# B&R Automation Studio project AutoCon2021 (part 2)

### GlobalTypes.typ
```iecst
(*Main System Interface Types*)

TYPE
	MainIfTyp : 	STRUCT
		Cmd : MainIfCmdTyp;
		Par : MainIfParTyp;
		Cfg : MainIfCfgTyp;
		Status : MainIfStatusTyp;
	END_STRUCT;
	MainIfCmdTyp : 	STRUCT
		Power : BOOL;
		Start : BOOL;
		Stop : BOOL;
		Reset : BOOL;
	END_STRUCT;
	MainIfParTyp : 	STRUCT
		Tmp : USINT;
	END_STRUCT;
	MainIfCfgTyp : 	STRUCT
		ShuttleCount : USINT;
	END_STRUCT;
	MainIfStatusTyp : 	STRUCT
		PowerOn : BOOL;
		Running : BOOL;
		Error : BOOL;
	END_STRUCT;
END_TYPE

(*Process Info Interface*)

TYPE
	ProcessInfoIfTyp : 	STRUCT
		Cmd : ProcessInfoIfCmdTyp;
		Par : ProcessInfoIfParTyp;
		Sts : ProcessInfoIfStsTyp;
	END_STRUCT;
	ProcessInfoIfCmdTyp : 	STRUCT
		Enable : BOOL;
		ResetData : BOOL;
	END_STRUCT;
	ProcessInfoIfParTyp : 	STRUCT
		CurrentProductCount : UDINT;
		CurrentPowderCount : UDINT;
	END_STRUCT;
	ProcessInfoIfStsTyp : 	STRUCT
		Enabled : BOOL;
		CurrentPPM : REAL;
		CurrentPPH : REAL;
		CurrentBlistersPerMinute : REAL;
		CurrentLayersPerMinute : REAL;
	END_STRUCT;
END_TYPE

(*Shuttle Interface Types*)

TYPE
	gShuttleIfTyp : 	STRUCT  (*Interface for controlling a shuttle*)
		Cmd : gShuttleIfCmdTyp; (*Commands to issue to a shuttle*)
		Par : gShuttleIfParTyp; (*Parameters for the process for this shuttle*)
		Cfg : gShuttleIfConfigTyp; (*Configuration values for this shuttle*)
		Flags : USINT;
		Status : gShuttleIfStatusTyp; (*Status information related to this shuttle*)
	END_STRUCT;
	gShuttleIfCmdTyp : 	STRUCT  (*Commands for controlling a shuttle*)
		Enable : BOOL; (*Command for enabling the control of a shuttle in the process*)
		Recover : BOOL; (*Command for a shuttle to start recovery*)
		NextStep : BOOL; (*Command for a shuttle to start the next step in the process*)
		ResetProductInfo : BOOL; (*Command to reset all the product info on a shuttle*)
		Stop : BOOL; (*Command to stop the process for a shuttle*)
	END_STRUCT;
	gShuttleIfParTyp : 	STRUCT  (*Parameters for the shuttle's operation*)
		NumLayers : USINT; (*Number of layers for this defined recipe*)
		MacroIDs : gShuttleIfCfgMacrosTyp; (*Macro's used for routing shuttles*)
	END_STRUCT;
	gShuttleIfCfgMacrosTyp : 	STRUCT  (*Structure of the macro IDs used for operation*)
		LoadToPrintMacroID : gShuttleIfMacroEnum; (*Macro ID used for sending a shuttle from the load station to the print station*)
		PrintToDoseMacroID : gShuttleIfMacroEnum; (*Macro ID used for sending a shuttle from the print station to the Dose station*)
		DoseToPrintMacroID : gShuttleIfMacroEnum; (*Macro ID used for sending a shuttle from the dosing station to the printing station*)
		PrintToTampMacroID : gShuttleIfMacroEnum; (*Macro ID used for sending a shuttle from the printing station to the tamping station*)
		TampToUnloadMacroID : gShuttleIfMacroEnum; (*Macro ID used for sending a shuttle from the tamping station to the unload station*)
		UnloadToLoadMacroID : gShuttleIfMacroEnum; (*Macro ID used for sending a shuttle from the unloading station to the loading station*)
	END_STRUCT;
	gShuttleIfConfigTyp : 	STRUCT  (*Configuration values for a shuttle*)
		ShuttleId : USINT; (*ShuttleID of this shuttle*)
	END_STRUCT;
	gShuttleIfStatusTyp : 	STRUCT  (*Status information for the shuttle*)
		CurrentDestination : gShuttleIfDestEnum; (*Destination the shuttle is currently moving towards*)
		BlisterPresent : BOOL; (*Status flag to denote that a blister pack has been loaded on the shuttle*)
		ProductTamped : BOOL; (*Status flag to denote that the product has  been tamped*)
		CurrentLayer : USINT; (*Current Layer being built on the shuttle*)
		ShuttleInfo : Acp6DShuttleInfoType; (*CurrentStatus Information about the shuttle*)
		Error : BOOL; (*Shuttle is currently in an error state*)
		ErrorState : ShStateEnum; (*State the shuttle errored at*)
		Recovered : BOOL; (*Shuttle has been recovered*)
	END_STRUCT;
	gShuttleIfMacroEnum :
		( (*Macro IDs that are used to denote which macro means what*)
		MACRO_LOAD_TO_PRINT := 128, (*Macro ID used for sending a shuttle from the load station to the print station*)
		MACRO_PRINT_TO_DOSE1, (*Macro ID for moving from the print station to the dose 1 station*)
		MACRO_PRINT_TO_DOSE2, (*Macro ID for moving from the print station to the dose 2 station*)
		MACRO_DOSE_TO_PRINT, (*Macro ID used for sending a shuttle from the dosing station to the printing station*)
		MACRO_PRINT_TO_TAMP, (*Macro ID used for sending a shuttle from the printing station to the tamping station*)
		MACRO_TAMP_TO_UNLOAD, (*Macro ID used for sending a shuttle from the tamping station to the unload station*)
		MACRO_UNLOAD_TO_LOAD, (*Macro ID used for sending a shuttle from the unloading station to the loading station*)
		MACRO_RECOVERY_GROUP0, (*Macro ID used for recovering the group 0 shuttles*)
		MACRO_RECOVERY_GROUP1, (*Macro ID used for recovering the group 1 shuttles*)
		MACRO_RECOVERY_GROUP2 (*Macro ID used for recovering the group 2 shuttles*)
		);
	gShuttleIfDestEnum :
		( (*Destinations for a shuttle to move to*)
		DEST_LOAD, (*Destination Load station*)
		DEST_PRINT, (*Destination Printing station*)
		DEST_DOSE1, (*Destination Dose 1 station*)
		DEST_DOSE2, (*Destination Dose 2 station*)
		DEST_TAMP, (*Destination Tamping station*)
		DEST_UNLOAD (*Destination unload*)
		);
	ShStateEnum :
		(
		SH_OFF, (*Shuttle is in the off/idle state*)
		SH_INIT, (*Shuttle is in the initilization state*)
		SH_STARTUP, (*Shuttle is in the startup state*)
		SH_IDLE, (*Shuttle is in the idle state after having been recovered*)
		SH_MOVE_TO_LOAD, (*Shuttle is moving to the load position*)
		SH_LOAD, (*Shuttle is currently being loaded*)
		SH_MOVE_TO_PRINT, (*Shuttle is moving to the print position*)
		SH_PRINT, (*Shuttle is currently being printed*)
		SH_DECIDE_DOSE, (*Shuttle is deciding which dose station to send the shuttle to*)
		SH_MOVE_TO_DOSE, (*Shuttle is moving towards the defined dosing station*)
		SH_DOSE, (*Shuttle is currently going through the dosing procedure*)
		SH_MOVE_TO_TAMP, (*Shuttle is moving to the tamping location*)
		SH_TAMP, (*Shuttle is currently being tamped*)
		SH_MOVE_TO_OFFLOAD, (*Shuttle is moving to the offload position*)
		SH_OFFLOAD, (*Shuttle is currently being offloaded*)
		SH_ERROR := 65535 (*Shuttle is in the error state*)
		);
END_TYPE

(*6D Controller Interface Types*)

TYPE
	Acp6DCmdType : 	STRUCT
		Power : BOOL;
		ErrorReset : BOOL;
		GetErrorInfo : BOOL;
	END_STRUCT;
	Acp6DCtrlType : 	STRUCT
		Cmd : Acp6DCmdType;
		Status : Acp6DStatusType;
		Par : Acp6DParType;
	END_STRUCT;
	Acp6DParType : 	STRUCT
		Mode : McAcp6DMoveModeEnum;
		PathType : McAcp6DInPlaneMovePathEnum;
		Acceleration : REAL;
		EndVelocity : REAL;
		Velocity : REAL;
		ShuttleID : USINT;
		SegmentID : USINT;
		PositionX : REAL;
		PositionY : REAL;
	END_STRUCT;
	Acp6DStatusType : 	STRUCT
		Error : BOOL;
		ErrorID : DINT;
		Ready : BOOL;
		PowerOn : BOOL;
		ReadyToPowerOn : BOOL;
		ErrorCodes : ARRAY[0..8]OF DINT;
	END_STRUCT;
	Acp6DShuttleInfoType : 	STRUCT
		State : Acp6DShuttleStateInfoTyp;
		Force : Acp6DShuttleForceInfoTyp;
		Position : Acp6DShuttlePosInfoTyp;
	END_STRUCT;
	Acp6DShuttleStateInfoTyp : 	STRUCT
		Valid : BOOL;
		Value : McAcp6DShuttleStateEnum;
	END_STRUCT;
	Acp6DShuttlePosInfoTyp : 	STRUCT
		Valid : BOOL;
		Value : McAcp6DShPositionInfoType;
	END_STRUCT;
	Acp6DShuttleForceInfoTyp : 	STRUCT
		Valid : BOOL;
		Value : McAcp6DShForceInfoType;
	END_STRUCT;
END_TYPE

(*Recovery Interface Type*)

TYPE
	Acp6DRecoveryIfTyp : 	STRUCT
		Cmd : Acp6DRecoveryCmdTyp;
		Par : Acp6DRecoveryParTyp;
		Sts : Acp6DRecoveryStsTyp;
	END_STRUCT;
	Acp6DRecoveryCmdTyp : 	STRUCT
		Recover : BOOL;
		Reset : BOOL;
	END_STRUCT;
	Acp6DRecoveryParTyp : 	STRUCT
		AutoDrivePositions : ARRAY[0..MAX_SHUTTLE_COUNT_ARRAY]OF Acp6DAutoDrivePosTyp;
		Vel : REAL;
		Accel : REAL;
	END_STRUCT;
	Acp6DRecoveryStsTyp : 	STRUCT
		Recovering : BOOL;
		ReadyToStartProc : BOOL;
		Done : BOOL;
		ShuttlesRecovered : BOOL;
		Error : BOOL;
	END_STRUCT;
	Acp6DAutoDrivePosTyp : 	STRUCT
		ShIdx : USINT;
		GroupNum : USINT; (*Group ID used for recovery. Lower group, lower priority*)
		X : REAL;
		Y : REAL;
	END_STRUCT;
END_TYPE

(***********************Station Types*)

TYPE
	StationIfTyp : 	STRUCT
		Cmd : StationIfCmdTyp; (*Commands to a station*)
		Par : {REDUND_UNREPLICABLE} UDINT; (*Address of the parameter structure*)
		Cfg : StationIfCfgTyp; (*Configuration values for the station*)
		Sts : StationIfStsTyp; (*Status of the station*)
	END_STRUCT;
	StationIfCmdTyp : 	STRUCT
		Enable : BOOL; (*Enables the process station*)
		Process : BOOL; (*Start a process for the station with the defined shuttle index*)
		Reset : BOOL; (*Resets the process from an any state*)
	END_STRUCT;
	StationIfCfgTyp : 	STRUCT
		StationPos : StationPositionTyp; (*Station's center world position*)
	END_STRUCT;
	StationIfStsTyp : 	STRUCT
		Enabled : BOOL; (*Signal denoting the station is enabled and in an operational state*)
		Processing : BOOL; (*Signal denoting the station is currently operating on a shuttle*)
		Done : BOOL; (*Signal denoting the current operation has completed*)
		ReadyForNewShuttle : BOOL; (*Signal denoting the station is ready for a new shuttle*)
		Error : BOOL; (*Signal denoting the station has an error present*)
	END_STRUCT;
END_TYPE

(*Load Station Types*)

TYPE
	LoadStationIfTyp : 	STRUCT
		Cmd : LoadStationCmdTyp; (*Commands to the station*)
		Par : LoadStationParTyp; (*Paramters for the station's operation*)
		Cfg : LoadStationCfgTyp; (*Configuration values for the station*)
		Status : LoadStationStatusTyp; (*Status of the station*)
	END_STRUCT;
	LoadStationCmdTyp : 	STRUCT
		Enable : BOOL; (*Enables the process station*)
		Process : BOOL; (*Start a process for the station with the defined shuttle index*)
		Reset : BOOL; (*Resets the process from an any state*)
	END_STRUCT;
	LoadStationParTyp : 	STRUCT
		ShuttleIdx : USINT; (*Index in the gShuttle array for the shuttle in question*)
		WaitTime : TIME; (*Amount of time to wait for the load process*)
	END_STRUCT;
	LoadStationCfgTyp : 	STRUCT
		StationPos : StationPositionTyp; (*Station's center world position*)
	END_STRUCT;
	LoadStationStatusTyp : 	STRUCT
		Enabled : BOOL; (*Signal denoting the station is enabled and in an operational state*)
		Processing : BOOL; (*Signal denoting the station is currently operating on a shuttle*)
		Done : BOOL; (*Signal denoting the current operation has completed*)
		ReadyForNewShuttle : BOOL; (*Signal denoting the station is ready for a new shuttle*)
		Error : BOOL; (*Signal denoting the station has an error present*)
	END_STRUCT;
	StationPositionTyp : 	STRUCT
		X : REAL; (*Station's Global X position*)
		Y : REAL; (*Station's Global Y position*)
	END_STRUCT;
END_TYPE

(*Unload Station Types*)

TYPE
	UnloadStationIfTyp : 	STRUCT
		Cmd : UnloadStationCmdTyp; (*Commands to the station*)
		Par : UnloadStationParTyp; (*Paramters for the station's operation*)
		Cfg : UnloadStationCfgTyp; (*Configuration values for the station*)
		Status : UnloadStationStatusTyp; (*Status of the station*)
	END_STRUCT;
	UnloadStationCmdTyp : 	STRUCT
		Enable : BOOL; (*Enables the process station*)
		Process : BOOL; (*Start a process for the station with the defined shuttle index*)
		Reset : BOOL; (*Resets the process from an any state*)
	END_STRUCT;
	UnloadStationParTyp : 	STRUCT
		ShuttleIdx : USINT; (*Index in the gShuttle array for the shuttle in question*)
		WaitTime : TIME; (*Amount of time to wait for the load process*)
	END_STRUCT;
	UnloadStationCfgTyp : 	STRUCT
		StationPos : StationPositionTyp; (*Station's center world position*)
	END_STRUCT;
	UnloadStationStatusTyp : 	STRUCT
		Enabled : BOOL; (*Signal denoting the station is enabled and in an operational state*)
		Processing : BOOL; (*Signal denoting the station is currently operating on a shuttle*)
		Done : BOOL; (*Signal denoting the current operation has completed*)
		ReadyForNewShuttle : BOOL; (*Signal denoting the station is ready for a new shuttle*)
		Error : BOOL; (*Signal denoting the station has an error present*)
	END_STRUCT;
END_TYPE

(*Print Station Types*)

TYPE
	PrintStationIfTyp : 	STRUCT
		Cmd : PrintStationCmdTyp; (*Commands to the station*)
		Par : PrintStationParTyp; (*Paramters for the station's operation*)
		Cfg : PrintStationCfgTyp; (*Configuration values for the station*)
		Status : PrintStationStatusTyp; (*Status of the station*)
	END_STRUCT;
	PrintStationCmdTyp : 	STRUCT
		Enable : BOOL; (*Enables the process station*)
		Process : BOOL; (*Start a process for the station with the defined shuttle index*)
		Reset : BOOL; (*Resets the process from an any state*)
	END_STRUCT;
	PrintStationParTyp : 	STRUCT
		ShuttleIdx : USINT; (*Index in the gShuttle array for the shuttle in question*)
		PrintVel : REAL; (*Speed at which to complete the print process m/s*)
		PrintEndVel : REAL; (*Speed at which the shuttle should end the print process at m/s*)
		PrintDistanceX : REAL; (*Distance for how far the print movement will go in the X direction (m)*)
		PrintDistanceY : REAL; (*Distance for how far the print movement will go in the Y direction(m)*)
		PrintAccel : REAL; (*Acceleration at which to use for the print process m/s2*)
	END_STRUCT;
	PrintStationCfgTyp : 	STRUCT
		StationPos : StationPositionTyp; (*Station's center world position*)
	END_STRUCT;
	PrintStationStatusTyp : 	STRUCT
		Enabled : BOOL; (*Signal denoting the station is enabled and in an operational state*)
		ReadyForNewShuttle : BOOL; (*Signal denoting the station is ready for a new shuttle*)
		Processing : BOOL; (*Signal denoting the station is currently operating on a shuttle*)
		Done : BOOL; (*Signal denoting the current operation has completed*)
		Error : BOOL; (*Signal denoting the station has an error present*)
	END_STRUCT;
END_TYPE

(*Dose Station Types*)

TYPE
	DoseStationIfTyp : 	STRUCT
		Cmd : DoseStationCmdTyp; (*Commands to the station*)
		Par : DoseStationParTyp; (*Paramters for the station's operation*)
		Cfg : DoseStationCfgTyp; (*Configuration values for the station*)
		Status : DoseStationStatusTyp; (*Status of the station*)
	END_STRUCT;
	DoseStationCmdTyp : 	STRUCT
		Enable : BOOL; (*Enables the process station*)
		Process : BOOL; (*Start a process for the station with the defined shuttle index*)
		Reset : BOOL; (*Resets the process from an any state*)
	END_STRUCT;
	DoseStationParTyp : 	STRUCT
		ShuttleIdx : USINT; (*Index in the gShuttle array for the shuttle in question*)
		Vel : REAL; (*Velocity to move for the defined index movement*)
		EndVel : REAL; (*Velocity to end the movement at for the defined index movement*)
		Accel : REAL; (*Acceleration to use for the defined index movement*)
		WaitTime : TIME; (*Time needed to preform each dose process*)
		NumRowsOfCavities : USINT; (*Number of rows of the cavities in the blister pack. Will be indexing this many times in the dosing process*)
		SpaceBetweenCavities : DoseIndexMovParsTyp; (*Space between cavities to index through*)
		FirstCavityPosition : DoseIndexMovParsTyp; (*Offset in m for the first cavity*)
	END_STRUCT;
	DoseStationCfgTyp : 	STRUCT
		StationPos : StationPositionTyp; (*Station's center world position*)
	END_STRUCT;
	DoseStationStatusTyp : 	STRUCT
		Enabled : BOOL; (*Signal denoting the station is enabled and in an operational state*)
		ReadyForNewShuttle : BOOL; (*Signal denoting the station is ready for a new shuttle*)
		Processing : BOOL; (*Signal denoting the station is currently operating on a shuttle*)
		Done : BOOL; (*Signal denoting the current operation has completed*)
		Error : BOOL; (*Signal denoting the station has an error present*)
	END_STRUCT;
	DoseIndexMovParsTyp : 	STRUCT
		DistX : REAL; (*Relative distance in X to move for a defined index (m)*)
		DistY : REAL; (*Relative distance in Y to move for a defined index (m)*)
	END_STRUCT;
END_TYPE

(*Tamp Station Types*)

TYPE
	TampStationIfTyp : 	STRUCT
		Cmd : TampStationCmdTyp; (*Commands to the station*)
		Par : TampStationParTyp; (*Paramters for the station's operation*)
		Cfg : TampStationCfgTyp; (*Configuration values for the station*)
		Status : TampStationStatusTyp; (*Status of the station*)
	END_STRUCT;
	TampStationCmdTyp : 	STRUCT
		Enable : BOOL; (*Enables the process station*)
		Process : BOOL; (*Start a process for the station with the defined shuttle index*)
		Reset : BOOL; (*Resets the process from an any state*)
	END_STRUCT;
	TampStationParTyp : 	STRUCT
		ShuttleIdx : USINT; (*Index in the gShuttle array for the shuttle in question*)
		EntranceMovement : TampMovementParTyp; (*Relative position to enter the tamp position*)
		ExitMovement : TampMovementParTyp; (*Relative positions to exit the tamp position*)
		TampHeight : REAL; (*Height in which to preform the z movement for the tamp process (m)*)
		Vel : REAL; (*Velocity to move for the defined index movement*)
		EndVel : REAL; (*Velocity to end the movement at for the defined index movement*)
		Accel : REAL; (*Acceleration to use for the defined index movement*)
		WaitTime : TIME; (*Time needed to preform each dose process*)
	END_STRUCT;
	TampStationCfgTyp : 	STRUCT
		StationPos : StationPositionTyp; (*Station's center world position*)
	END_STRUCT;
	TampStationStatusTyp : 	STRUCT
		Enabled : BOOL; (*Signal denoting the station is enabled and in an operational state*)
		ReadyForNewShuttle : BOOL; (*Signal denoting the station is ready for a new shuttle*)
		Processing : BOOL; (*Signal denoting the station is currently operating on a shuttle*)
		Done : BOOL; (*Signal denoting the current operation has completed*)
		Error : BOOL; (*Signal denoting the station has an error present*)
	END_STRUCT;
	TampMovementParTyp : 	STRUCT
		DistX : REAL; (*Relative distance in X to move for a defined movement(m)*)
		DistY : REAL; (*Relative distance in Y to move for a defined movement(m)*)
	END_STRUCT;
END_TYPE
```

### Package Logical/Source/ShuttleCtrl - Package that contains code for controlling individual shuttles

### Program Logical/Source/ShuttleCtrl/ShCtrl (IEC)

#### Cyclic.st - Cyclic code
```iecst
PROGRAM _CYCLIC
	FOR i:= 0 TO gMainIf.Cfg.ShuttleCount - 1 DO

		IF gShuttleIf[i].Status.CurrentDestination = DEST_DOSE1 THEN
			pDoseStationIf ACCESS ADR(gDoseStationsIf[0]);
		ELSIF gShuttleIf[i].Status.CurrentDestination = DEST_DOSE2 THEN
			pDoseStationIf ACCESS ADR(gDoseStationsIf[1]);
		END_IF

		CASE shState[i] OF
			SH_OFF:  //******************************************************************************** Shuttle is in the off/idle state
				IF gShuttleIf[i].Cmd.Enable THEN
					shState[i] := SH_INIT;
				ELSE

				END_IF
			SH_INIT:  //******************************************************************************** Shuttle is in the initilization state
				//In this state we could make any checks on the current shuttle process perhaps in order to aide in recovery?

				shState[i] := SH_STARTUP;
			SH_STARTUP:  //******************************************************************************** Shuttle is in the startup state
				//In this state maybe we have triggered recovery and we're waiting for the autodrive to complete
				shState[i] := SH_IDLE;
			SH_IDLE:  //******************************************************************************** Shuttle is in the idle state
				IF gShuttleIf[i].Cmd.NextStep THEN
					gShuttleIf[i].Cmd.NextStep := FALSE;
					//Evaluate the current step to determine what the next step should be
					shFbs[i].ShRunMacroFb.Controller := ADR(gMcAcp6DController);
					shFbs[i].ShRunMacroFb.ShuttleID := gShuttleIf[i].Cfg.ShuttleId;
					shFbs[i].ShRunMacroFb.MacroID := UDINT_TO_USINT(gShuttleIf[i].Par.MacroIDs.UnloadToLoadMacroID);
					shFbs[i].ShRunMacroFb.Execute := TRUE;
					gShuttleIf[i].Status.CurrentDestination := DEST_LOAD;
					LogDebug(gAuditTrail,i,"Sent to Load");
					//MpAuditCustomEvent(gAuditTrail,"INFO","Sh","Powered On");

					shState[i] := SH_MOVE_TO_LOAD;
				END_IF
			SH_MOVE_TO_LOAD:  //******************************************************************************** Shuttle is moving to the load position
				IF shFbs[i].ShRunMacroFb.Error THEN
					gShuttleIf[i].Status.Error := TRUE;
					gShuttleIf[i].Status.ErrorState := shState[i];
					shState[i] := SH_ERROR;
				ELSIF shFbs[i].ShRunMacroFb.Done AND (gLoadStationIf.Par.ShuttleIdx = STATION_IS_EMPTY AND gLoadStationIf.Status.ReadyForNewShuttle)
					AND PositionValidation(ADR(gLoadStationIf.Cfg.StationPos),ADR(gShuttleIf[i].Status.ShuttleInfo.Position)) THEN
					gLoadStationIf.Par.ShuttleIdx := i;
					gLoadStationIf.Cmd.Process := TRUE;

					LogDebug(gAuditTrail,i,"Arrived at Load");

					shFbs[i].ShRunMacroFb.Execute := FALSE;
					shState[i] := SH_LOAD;
				END_IF
			SH_LOAD:  //******************************************************************************** Shuttle is currently being loaded
				//Station has control on the shuttle during this section
				IF gShuttleIf[i].Cmd.NextStep THEN
					gLoadStationIf.Cmd.Process := FALSE; //Respond to the Load station we're done

					gShuttleIf[i].Status.BlisterPresent := TRUE;
					gShuttleIf[i].Cmd.NextStep := FALSE;
					gShuttleIf[i].Status.CurrentDestination := DEST_PRINT;

					shFbs[i].ShRunMacroFb.Controller := ADR(gMcAcp6DController);
					shFbs[i].ShRunMacroFb.ShuttleID := gShuttleIf[i].Cfg.ShuttleId;
					shFbs[i].ShRunMacroFb.MacroID := UDINT_TO_USINT(gShuttleIf[i].Par.MacroIDs.LoadToPrintMacroID);
					shFbs[i].ShRunMacroFb.Execute := TRUE;

					LogDebug(gAuditTrail,i,"Sent To Print");

					shState[i] := SH_MOVE_TO_PRINT;
				END_IF
			SH_MOVE_TO_PRINT:  //******************************************************************************** Shuttle is moving to the print position
				IF shFbs[i].ShRunMacroFb.Error THEN
					gShuttleIf[i].Status.Error := TRUE;
					gShuttleIf[i].Status.ErrorState := shState[i];
					shState[i] := SH_ERROR;
				ELSIF shFbs[i].ShRunMacroFb.Done AND (gPrintStationIf.Par.ShuttleIdx = STATION_IS_EMPTY AND gPrintStationIf.Status.ReadyForNewShuttle)
					AND PositionValidation(ADR(gPrintStationIf.Cfg.StationPos),ADR(gShuttleIf[i].Status.ShuttleInfo.Position)) THEN
					gPrintStationIf.Par.ShuttleIdx := i; //Replace with idx when adding the loop
					gPrintStationIf.Cmd.Process := TRUE;

					LogDebug(gAuditTrail,i,"Arrived at Print");

					shFbs[i].ShRunMacroFb.Execute := FALSE;
					shState[i] := SH_PRINT;
				END_IF
			SH_PRINT:  //******************************************************************************** Shuttle is currently being printed
				//Station has control on the shuttle during this section
				IF gShuttleIf[i].Cmd.NextStep THEN
					gPrintStationIf.Cmd.Process := FALSE; //Respond to the print station we're done

					gShuttleIf[i].Status.CurrentLayer :=  gShuttleIf[i].Status.CurrentLayer + 1;
					LogDebug(gAuditTrail,i,"Print complete");
					gShuttleIf[i].Cmd.NextStep := FALSE;

					shState[i] := SH_DECIDE_DOSE;
				END_IF
			SH_DECIDE_DOSE:  //******************************************************************************** Shuttle is deciding which dose station to send the shuttle to
				//First check if the layers have finished
				IF gShuttleIf[i].Status.CurrentLayer > gShuttleIf[i].Par.NumLayers THEN
					//We've finished layering move to the tamp state
					shFbs[i].ShRunMacroFb.Controller := ADR(gMcAcp6DController);
					shFbs[i].ShRunMacroFb.ShuttleID := gShuttleIf[i].Cfg.ShuttleId;
					shFbs[i].ShRunMacroFb.MacroID := UDINT_TO_USINT(gShuttleIf[i].Par.MacroIDs.PrintToTampMacroID);
					shFbs[i].ShRunMacroFb.Execute := TRUE;

					gShuttleIf[i].Status.CurrentDestination := DEST_TAMP;
					LogDebug(gAuditTrail,i,"Sent to Tamp");

					shState[i] := SH_MOVE_TO_TAMP;
				ELSE
					//Need to determine which doser is available
					IF NextDoseStation = DEST_DOSE1 THEN
						gShuttleIf[i].Par.MacroIDs.PrintToDoseMacroID := MACRO_PRINT_TO_DOSE1;
						gShuttleIf[i].Status.CurrentDestination := DEST_DOSE1;
						LogDebug(gAuditTrail,i,"Sent To Dose 1");
						NextDoseStation := DEST_DOSE2;
					ELSE
						gShuttleIf[i].Par.MacroIDs.PrintToDoseMacroID := MACRO_PRINT_TO_DOSE2;
						gShuttleIf[i].Status.CurrentDestination := DEST_DOSE2;
						LogDebug(gAuditTrail,i,"Sent To Dose 2");
						NextDoseStation := DEST_DOSE1;
					END_IF

					shFbs[i].ShRunMacroFb.Controller := ADR(gMcAcp6DController);
					shFbs[i].ShRunMacroFb.ShuttleID := gShuttleIf[i].Cfg.ShuttleId;
					shFbs[i].ShRunMacroFb.MacroID := UDINT_TO_USINT(gShuttleIf[i].Par.MacroIDs.PrintToDoseMacroID);
					shFbs[i].ShRunMacroFb.Execute := TRUE;

					shState[i] := SH_MOVE_TO_DOSE;
				END_IF
			SH_MOVE_TO_DOSE:  //******************************************************************************** Shuttle is moving towards the defined dosing station
				IF shFbs[i].ShRunMacroFb.Error THEN
					gShuttleIf[i].Status.Error := TRUE;
					gShuttleIf[i].Status.ErrorState := shState[i];
					shState[i] := SH_ERROR;
				ELSIF shFbs[i].ShRunMacroFb.Done AND (pDoseStationIf.Par.ShuttleIdx = STATION_IS_EMPTY AND pDoseStationIf.Status.ReadyForNewShuttle AND NOT pDoseStationIf.Cmd.Process)
					AND PositionValidation(ADR(pDoseStationIf.Cfg.StationPos),ADR(gShuttleIf[i].Status.ShuttleInfo.Position)) THEN//Wait for the movement to end and the Station to be ready to accept a new shuttle
					pDoseStationIf.Par.ShuttleIdx := i;
					pDoseStationIf.Cmd.Process := TRUE;

					LogDebug(gAuditTrail,i,"Arrived at Dose");

					shFbs[i].ShRunMacroFb.Execute := FALSE;
					shState[i] := SH_DOSE;
				END_IF
			SH_DOSE:  //******************************************************************************** Shuttle is currently going through the dosing procedure
				//Station has control on the shuttle during this section
				IF gShuttleIf[i].Cmd.NextStep THEN
					gShuttleIf[i].Cmd.NextStep := FALSE;
					pDoseStationIf.Cmd.Process := FALSE; //Respond to the dose station we're done

					gShuttleIf[i].Status.CurrentDestination := DEST_PRINT;

					shFbs[i].ShRunMacroFb.Controller := ADR(gMcAcp6DController);
					shFbs[i].ShRunMacroFb.ShuttleID := gShuttleIf[i].Cfg.ShuttleId;
					shFbs[i].ShRunMacroFb.MacroID := UDINT_TO_USINT(gShuttleIf[i].Par.MacroIDs.DoseToPrintMacroID);
					shFbs[i].ShRunMacroFb.Execute := TRUE;

					LogDebug(gAuditTrail,i,"Sent To Print");

					shState[i] := SH_MOVE_TO_PRINT;
				END_IF
			SH_MOVE_TO_TAMP:  //******************************************************************************** Shuttle is moving to the tamping location
				IF shFbs[i].ShRunMacroFb.Error THEN
					gShuttleIf[i].Status.Error := TRUE;
					gShuttleIf[i].Status.ErrorState := shState[i];
					shState[i] := SH_ERROR;
				ELSIF shFbs[i].ShRunMacroFb.Done AND (gTampStationIf.Par.ShuttleIdx = STATION_IS_EMPTY AND gTampStationIf.Status.ReadyForNewShuttle)
					AND PositionValidation(ADR(gTampStationIf.Cfg.StationPos),ADR(gShuttleIf[i].Status.ShuttleInfo.Position)) THEN
					gTampStationIf.Par.ShuttleIdx := i;
					gTampStationIf.Cmd.Process := TRUE;

					LogDebug(gAuditTrail,i,"Arrived at Tamp");

					shFbs[i].ShRunMacroFb.Execute := FALSE;
					shState[i] := SH_TAMP;
				END_IF
			SH_TAMP:  //******************************************************************************** Shuttle is currently being tamped
				//Station has control on the shuttle during this section
				IF gShuttleIf[i].Cmd.NextStep THEN
					gTampStationIf.Cmd.Process := FALSE;//Respond to the unload station we're done

					gShuttleIf[i].Status.ProductTamped := TRUE;
					gShuttleIf[i].Cmd.NextStep := FALSE;

					gShuttleIf[i].Status.CurrentDestination := DEST_UNLOAD;

					shFbs[i].ShRunMacroFb.Controller := ADR(gMcAcp6DController);
					shFbs[i].ShRunMacroFb.ShuttleID := gShuttleIf[i].Cfg.ShuttleId;
					shFbs[i].ShRunMacroFb.MacroID := UDINT_TO_USINT(gShuttleIf[i].Par.MacroIDs.TampToUnloadMacroID);
					shFbs[i].ShRunMacroFb.Execute := TRUE;

					LogDebug(gAuditTrail,i,"Sent To Unload");

					shState[i] := SH_MOVE_TO_OFFLOAD;
				END_IF
			SH_MOVE_TO_OFFLOAD:  //******************************************************************************** Shuttle is moving to the offload position
				IF shFbs[i].ShRunMacroFb.Error THEN
					gShuttleIf[i].Status.Error := TRUE;
					gShuttleIf[i].Status.ErrorState := shState[i];
					shState[i] := SH_ERROR;
				ELSIF shFbs[i].ShRunMacroFb.Done AND (gUnloadStationIf.Par.ShuttleIdx = STATION_IS_EMPTY AND gUnloadStationIf.Status.ReadyForNewShuttle)
					AND PositionValidation(ADR(gUnloadStationIf.Cfg.StationPos),ADR(gShuttleIf[i].Status.ShuttleInfo.Position)) THEN
					gUnloadStationIf.Par.ShuttleIdx := i;
					gUnloadStationIf.Cmd.Process := TRUE;

					LogDebug(gAuditTrail,i,"Arrived at unload");

					shFbs[i].ShRunMacroFb.Execute := FALSE;
					shState[i] := SH_OFFLOAD;
				END_IF
			SH_OFFLOAD:  //******************************************************************************** Shuttle is currently being offloaded
				//Station has control on the shuttle during this section
				IF gShuttleIf[i].Cmd.NextStep THEN
					gUnloadStationIf.Cmd.Process := FALSE; //Respond to the unload station we're done

					gShuttleIf[i].Cmd.NextStep := FALSE;
					gShuttleIf[i].Cmd.ResetProductInfo := TRUE;
					gShuttleIf[i].Status.CurrentDestination := DEST_LOAD;

					//Increment the process counter
					gProcessInfoIf.Par.CurrentProductCount := gProcessInfoIf.Par.CurrentProductCount + 1;

					IF gShuttleIf[i].Cmd.Stop THEN
						gShuttleIf[i].Cmd.Stop := FALSE;
						shState[i] := SH_INIT;
					ELSE
						shFbs[i].ShRunMacroFb.Controller := ADR(gMcAcp6DController);
						shFbs[i].ShRunMacroFb.ShuttleID := gShuttleIf[i].Cfg.ShuttleId;
						shFbs[i].ShRunMacroFb.MacroID := UDINT_TO_USINT(gShuttleIf[i].Par.MacroIDs.UnloadToLoadMacroID);
						shFbs[i].ShRunMacroFb.Execute := TRUE;

						LogDebug(gAuditTrail,i,"Sent To Load");

						shState[i] := SH_MOVE_TO_LOAD;
					END_IF

				END_IF
			SH_ERROR: //******************************************************************************** Shuttle is in the error state

		END_CASE;
		shFbs[i].ShRunMacroFb();

		IF gShuttleIf[i].Cmd.ResetProductInfo THEN
			gShuttleIf[i].Status.CurrentDestination := DEST_LOAD;
			gShuttleIf[i].Status.BlisterPresent := FALSE;
			gShuttleIf[i].Status.CurrentLayer := 0;
			gShuttleIf[i].Status.Error := FALSE;
			gShuttleIf[i].Status.ErrorState := 0;
			gShuttleIf[i].Status.ProductTamped := 0;
			gShuttleIf[i].Cmd.ResetProductInfo := FALSE;
		END_IF
	END_FOR;
	pDebugIf ACCESS ADR(gShuttleIf[debugIdx]);
	pDebugState ACCESS ADR(shState[debugIdx]);
	pDebugFbs ACCESS ADR(shFbs[debugIdx]);

END_PROGRAM
```

#### Init.st - Init code
```iecst
PROGRAM _INIT
	FOR i:=0 TO MAX_SHUTTLE_COUNT-1 DO
		gShuttleIf[i].Par.MacroIDs.LoadToPrintMacroID := MACRO_LOAD_TO_PRINT;
		gShuttleIf[i].Par.MacroIDs.PrintToTampMacroID := MACRO_PRINT_TO_TAMP;
		gShuttleIf[i].Par.MacroIDs.PrintToDoseMacroID := MACRO_PRINT_TO_DOSE2; //Hard coding this for now
		gShuttleIf[i].Par.MacroIDs.DoseToPrintMacroID:= MACRO_DOSE_TO_PRINT;
		gShuttleIf[i].Par.MacroIDs.TampToUnloadMacroID := MACRO_TAMP_TO_UNLOAD;
		gShuttleIf[i].Par.MacroIDs.UnloadToLoadMacroID := MACRO_UNLOAD_TO_LOAD;
		//The print to dose is defined in the shuttle decide dose task

		gShuttleIf[i].Par.NumLayers := 4;
	END_FOR;

	NextDoseStation := DEST_DOSE1;
END_PROGRAM
```

#### Types.typ - Local data types
```iecst
TYPE
	ShFbsTyp : 	STRUCT
		ShRunMacroFb : MC_BR_MacroRun_Acp6D; (*Execute a macro on the current shuttle*)
	END_STRUCT;
	ShCycleIfs : {REDUND_UNREPLICABLE} 	STRUCT
		Dose : REFERENCE TO DoseStationIfTyp;
	END_STRUCT;
END_TYPE
```

#### Variables.var - Local variables
```iecst
VAR
	i : USINT; (*Loop index*)
	shState : ARRAY[0..MAX_SHUTTLE_COUNT_ARRAY] OF ShStateEnum;
	shFbs : ARRAY[0..MAX_SHUTTLE_COUNT_ARRAY] OF ShFbsTyp;
	stationIfs : {REDUND_UNREPLICABLE} ARRAY[0..MAX_SHUTTLE_COUNT_ARRAY] OF ShCycleIfs;
	NextDoseStation : gShuttleIfDestEnum;
	pDoseStationIf : REFERENCE TO DoseStationIfTyp;
	pDebugIf : REFERENCE TO gShuttleIfTyp;
	pDebugFbs : REFERENCE TO ShFbsTyp;
	pDebugState : REFERENCE TO ShStateEnum;
	debugIdx : USINT;
END_VAR
```

#### LocalFunctions.fun
```iecst
FUNCTION LogDebug : USINT
	VAR_INPUT
		MpLink : MpComIdentType;
		Idx : USINT;
		Msg : WSTRING[100];
	END_VAR
	VAR
		msg : WSTRING[100];
		typ : WSTRING[100];
	END_VAR
END_FUNCTION

{REDUND_ERROR} FUNCTION PositionValidation : BOOL (*Validates if a shuttle is in the defined position*) (*$GROUP=User,$CAT=User,$GROUPICON=User.png,$CATICON=User.png*)
	VAR_INPUT
		DestinationPosition : REFERENCE TO StationPositionTyp;
		CurrentInfo : REFERENCE TO Acp6DShuttlePosInfoTyp;
	END_VAR
END_FUNCTION
```

#### PositionValidation.st
```iecst
(* Validates if a shuttle is in the defined position *)
FUNCTION PositionValidation
	IF CurrentInfo.Valid THEN
		IF CurrentInfo.Value.X >= DestinationPosition.X - 0.00001
			AND CurrentInfo.Value.X <= DestinationPosition.X + 0.00001
			AND CurrentInfo.Value.Y >= DestinationPosition.Y - 0.00001
			AND CurrentInfo.Value.Y <= DestinationPosition.Y + 0.00001 THEN
			PositionValidation := TRUE;
		ELSE
			PositionValidation := FALSE;
		END_IF

	ELSE
		PositionValidation := FALSE;
	END_IF
END_FUNCTION

FUNCTION LogDebug
	msg := "";
	typ := "Sh ";
	typ := USINT_TO_WSTRING(Idx);
	MpAuditCustomEvent(MpLink,"DEBUG",typ,Msg);
END_FUNCTION
```

#### LocalFunctions.st - not listed in the package file held
```iecst
(* Validates if a shuttle is in the defined position *)
FUNCTION PositionValidation
	IF CurrentInfo.Valid THEN
		IF CurrentInfo.Value.X >= DestinationPosition.X - 0.00001
			AND CurrentInfo.Value.X <= DestinationPosition.X + 0.00001
			AND CurrentInfo.Value.Y >= DestinationPosition.Y - 0.00001
			AND CurrentInfo.Value.Y <= DestinationPosition.Y + 0.00001 THEN
			PositionValidation := TRUE;
		ELSE
			PositionValidation := FALSE;
		END_IF

	ELSE
		PositionValidation := FALSE;
	END_IF
END_FUNCTION

FUNCTION LogDebug
	msg := "";
	typ := "Sh ";
	typ := USINT_TO_WSTRING(Idx);
	MpAuditCustomEvent(MpLink,"DEBUG",typ,Msg);
END_FUNCTION

FUNCTION BufferCount
	LaneCounts[0] := 0;
	LaneCounts[1] := 0;
	LaneCounts[2] := 0;
	FOR i:=0 TO ShuttleCnt - 1 DO
		IF Shuttles[i].Sts.ProductInfo.Buffer THEN
			LaneCounts[Shuttles[i].Sts.ProductInfo.BufferLane] := LaneCounts[Shuttles[i].Sts.ProductInfo.BufferLane] + 1;
		END_IF
	END_FOR;
END_FUNCTION

FUNCTION GetNextLane
	lowestCount := 255;
	FOR i := 0 TO 2 DO
		IF LaneCounts[i] < lowestCount THEN
			lowestCount := LaneCounts[i];
			curLane := i;
		END_IF
	END_FOR
	GetNextLane := curLane;
END_FUNCTION
```

### Program Logical/Source/ShuttleCtrl/Recovery (IEC)

#### Types.typ
```iecst
TYPE
	RecoveryFbs : 	STRUCT
		AsyncMoveFb : MC_BR_MoveInPlaneAsync_Acp6D;
		MacroRunFb : ARRAY[0..MAX_SHUTTLE_COUNT_ARRAY]OF MC_BR_MacroRun_Acp6D;
	END_STRUCT;
	RecoveryStateEnum :
		(
		RECOVER_IDLE, (*Recovery is in an idle state*)
		RECOVER_INIT, (*Initalize recovery state*)
		RECOVER_AUTODRIVE, (*Preform autodrive movement for recovery*)
		RECOVER_WAIT_ALL_RECOVER, (*Preform the loop through all shuttles to accomplish the reocvery*)
		RECOVER_DONE, (*Recovery has been completed*)
		RECOVER_ERROR (*Recovery had an error*)
		);
END_TYPE
```

#### Variables.var
```iecst
VAR
	CurrentGroup : USINT;
	GroupRecovered : BOOL;
	state : RecoveryStateEnum;
	RecoverFbs : RecoveryFbs;
END_VAR
VAR CONSTANT
	NUM_GROUPS : USINT := 3;
END_VAR
VAR
	i : USINT;
END_VAR
```

#### Cyclic.st
```iecst
PROGRAM _CYCLIC

	(*
	Shuttle reocvery
		Move all shuttles to autodrive positions
		Wait for autodrive to be finished
		loop through each shuttle
			if that shuttle's group is current
				it is not recovered,
					groupRecovered=false
					Evaluate each shuttle's position
					Send it to the unload position and set the "Next step cmd" to be true
				else
					onwards, do nothing

	*)

	CASE state OF
		RECOVER_IDLE:   //******************************************************************************** Recovery is in an idle state*)
			IF g6DRecoveryIf.Cmd.Recover THEN
				g6DRecoveryIf.Sts.Recovering := TRUE;
				state := RECOVER_INIT;
			END_IF
		RECOVER_INIT:   //******************************************************************************** Initalize recovery state*)
			RecoverFbs.AsyncMoveFb.Controller := ADR(gMcAcp6DController);
			RecoverFbs.AsyncMoveFb.NumberOfShuttles := gMainIf.Cfg.ShuttleCount;
			RecoverFbs.AsyncMoveFb.Velocity := g6DRecoveryIf.Par.Vel;
			RecoverFbs.AsyncMoveFb.Acceleration := g6DRecoveryIf.Par.Accel;
			FOR i:=0 TO gMainIf.Cfg.ShuttleCount - 1 DO
				RecoverFbs.AsyncMoveFb.PositionX[i] := g6DRecoveryIf.Par.AutoDrivePositions[i].X;
				RecoverFbs.AsyncMoveFb.PositionY[i] := g6DRecoveryIf.Par.AutoDrivePositions[i].Y;
				RecoverFbs.AsyncMoveFb.ShuttleID[i] := gShuttleIf[g6DRecoveryIf.Par.AutoDrivePositions[i].ShIdx].Cfg.ShuttleId;
				IF RecoverFbs.AsyncMoveFb.ShuttleID[i] = 0 THEN// Invalid shuttle id here
					g6DRecoveryIf.Sts.Error := TRUE;
				END_IF
			END_FOR;
			IF NOT g6DRecoveryIf.Sts.Error THEN
				RecoverFbs.AsyncMoveFb.Execute := TRUE;
				state := RECOVER_AUTODRIVE;
			ELSE
				state := RECOVER_ERROR;
			END_IF

		RECOVER_AUTODRIVE:   //******************************************************************************** Preform autodrive movement for recovery*)
			IF RecoverFbs.AsyncMoveFb.Error THEN
				g6DRecoveryIf.Sts.Error := TRUE;
				state := RECOVER_ERROR;
			ELSIF RecoverFbs.AsyncMoveFb.Done THEN
				g6DRecoveryIf.Sts.ReadyToStartProc := TRUE;
				RecoverFbs.AsyncMoveFb.Execute := FALSE;

				CurrentGroup := 0;
				state := RECOVER_WAIT_ALL_RECOVER;
			END_IF
		RECOVER_WAIT_ALL_RECOVER:   //******************************************************************************** Preform the loop through all shuttles to accomplish the reocvery*)
			//Ideally this should be in a FB
			GroupRecovered := TRUE;
			FOR i:=0 TO gMainIf.Cfg.ShuttleCount -1 DO
				IF g6DRecoveryIf.Par.AutoDrivePositions[i].GroupNum = CurrentGroup THEN
					IF NOT gShuttleIf[g6DRecoveryIf.Par.AutoDrivePositions[i].ShIdx].Status.Recovered THEN
						GroupRecovered := FALSE;
						IF CurrentGroup = 0 THEN
							gShuttleIf[g6DRecoveryIf.Par.AutoDrivePositions[i].ShIdx].Status.Recovered := TRUE;
							gShuttleIf[g6DRecoveryIf.Par.AutoDrivePositions[i].ShIdx].Cmd.NextStep := TRUE;
						ELSE
							RecoverFbs.MacroRunFb[i].Controller := ADR(gMcAcp6DController);
							RecoverFbs.MacroRunFb[i].MacroID := DINT_TO_USINT(MACRO_RECOVERY_GROUP0) + CurrentGroup;
							RecoverFbs.MacroRunFb[i].ShuttleID := gShuttleIf[g6DRecoveryIf.Par.AutoDrivePositions[i].ShIdx].Cfg.ShuttleId;
							RecoverFbs.MacroRunFb[i].Execute := TRUE;

							IF RecoverFbs.MacroRunFb[i].Error THEN
								g6DRecoveryIf.Sts.Error := TRUE;
							ELSIF RecoverFbs.MacroRunFb[i].Acknowledge THEN
								RecoverFbs.MacroRunFb[i].Execute := FALSE;
								gShuttleIf[g6DRecoveryIf.Par.AutoDrivePositions[i].ShIdx].Cmd.NextStep := TRUE;
								gShuttleIf[g6DRecoveryIf.Par.AutoDrivePositions[i].ShIdx].Status.Recovered := TRUE;
							END_IF
						END_IF
					ELSE
						//Already recovered don't have to do anything

					END_IF
				END_IF
			END_FOR;
			IF GroupRecovered THEN
				CurrentGroup := CurrentGroup + 1;
				IF CurrentGroup >= NUM_GROUPS THEN
					//We've recovered all groups
					g6DRecoveryIf.Sts.Recovering := FALSE;
					g6DRecoveryIf.Sts.Done := TRUE;
					g6DRecoveryIf.Sts.ShuttlesRecovered := TRUE;
					state := RECOVER_DONE;
				ELSE
					//Still more groups to recover, keep on recovering
				END_IF
			ELSE
				//Still more shuttles to recover in the group
			END_IF
			IF g6DRecoveryIf.Sts.Error THEN
				state := RECOVER_ERROR;
			END_IF
		RECOVER_DONE:   //******************************************************************************** Recovery has been completed*)
			IF NOT g6DRecoveryIf.Cmd.Recover THEN
				g6DRecoveryIf.Cmd.Reset := FALSE;
				g6DRecoveryIf.Sts.Done := FALSE;
				g6DRecoveryIf.Sts.ReadyToStartProc := FALSE;
				g6DRecoveryIf.Sts.Recovering := FALSE;
				g6DRecoveryIf.Sts.ShuttlesRecovered := FALSE;
				g6DRecoveryIf.Sts.Error := FALSE;
				CurrentGroup := 0;

				RecoverFbs.AsyncMoveFb.Execute := FALSE;
				state := RECOVER_IDLE;
			END_IF
		RECOVER_ERROR:   //******************************************************************************** Recovery had an error*)
			IF g6DRecoveryIf.Cmd.Reset THEN
				g6DRecoveryIf.Cmd.Reset := FALSE;
				g6DRecoveryIf.Sts.Done := FALSE;
				g6DRecoveryIf.Sts.ReadyToStartProc := FALSE;
				g6DRecoveryIf.Sts.Recovering := FALSE;
				g6DRecoveryIf.Sts.ShuttlesRecovered := FALSE;
				g6DRecoveryIf.Sts.Error := FALSE;
				CurrentGroup := 0;

				RecoverFbs.AsyncMoveFb.Execute := FALSE;
				state := RECOVER_IDLE;
			END_IF
	END_CASE;
	RecoverFbs.AsyncMoveFb();
	FOR i:=0 TO gMainIf.Cfg.ShuttleCount -1 DO
		RecoverFbs.MacroRunFb[i]();
	END_FOR;
END_PROGRAM
```

#### Init.st
```iecst
PROGRAM _INIT
	g6DRecoveryIf.Par.Vel := 1;
	g6DRecoveryIf.Par.Accel := 10;

	//************************************************************************* Shuttle 1
	g6DRecoveryIf.Par.AutoDrivePositions[0].ShIdx := 0;
	g6DRecoveryIf.Par.AutoDrivePositions[0].GroupNum := 0;
	g6DRecoveryIf.Par.AutoDrivePositions[0].X := 0.06;
	g6DRecoveryIf.Par.AutoDrivePositions[0].Y := 0.3;
	//************************************************************************* Shuttle 2
	g6DRecoveryIf.Par.AutoDrivePositions[1].ShIdx := 1;
	g6DRecoveryIf.Par.AutoDrivePositions[1].GroupNum := 1;
	g6DRecoveryIf.Par.AutoDrivePositions[1].X := 0.06;
	g6DRecoveryIf.Par.AutoDrivePositions[1].Y := 0.42;
	//************************************************************************* Shuttle 3
	g6DRecoveryIf.Par.AutoDrivePositions[2].ShIdx := 2;
	g6DRecoveryIf.Par.AutoDrivePositions[2].GroupNum := 1;
	g6DRecoveryIf.Par.AutoDrivePositions[2].X := 0.18;
	g6DRecoveryIf.Par.AutoDrivePositions[2].Y := 0.42;
	//************************************************************************* Shuttle 4
	g6DRecoveryIf.Par.AutoDrivePositions[3].ShIdx := 3;
	g6DRecoveryIf.Par.AutoDrivePositions[3].GroupNum := 1;
	g6DRecoveryIf.Par.AutoDrivePositions[3].X := 0.3;
	g6DRecoveryIf.Par.AutoDrivePositions[3].Y := 0.42;
	//************************************************************************* Shuttle 5
	g6DRecoveryIf.Par.AutoDrivePositions[4].ShIdx := 4;
	g6DRecoveryIf.Par.AutoDrivePositions[4].GroupNum := 1;
	g6DRecoveryIf.Par.AutoDrivePositions[4].X := 0.42;
	g6DRecoveryIf.Par.AutoDrivePositions[4].Y := 0.42;
	//************************************************************************* Shuttle 6
	g6DRecoveryIf.Par.AutoDrivePositions[5].ShIdx := 5;
	g6DRecoveryIf.Par.AutoDrivePositions[5].GroupNum := 1;
	g6DRecoveryIf.Par.AutoDrivePositions[5].X := 0.54;
	g6DRecoveryIf.Par.AutoDrivePositions[5].Y := 0.42;
	//************************************************************************* Shuttle 7
	g6DRecoveryIf.Par.AutoDrivePositions[6].ShIdx := 6;
	g6DRecoveryIf.Par.AutoDrivePositions[6].GroupNum := 1;
	g6DRecoveryIf.Par.AutoDrivePositions[6].X := 0.66;
	g6DRecoveryIf.Par.AutoDrivePositions[6].Y := 0.42;
	//************************************************************************* Shuttle 8
	g6DRecoveryIf.Par.AutoDrivePositions[7].ShIdx := 7;
	g6DRecoveryIf.Par.AutoDrivePositions[7].GroupNum := 2;
	g6DRecoveryIf.Par.AutoDrivePositions[7].X := 0.66;
	g6DRecoveryIf.Par.AutoDrivePositions[7].Y := 0.54;
END_PROGRAM
```

### Program Logical/Source/ProcessStations/LoadStation (IEC)

#### Types.typ
```iecst
TYPE
	LoadStationStateEnum :
		(
		LOAD_OFF, (*Load station is currently disabled*)
		LOAD_INIT, (*Load station is initalizing*)
		LOAD_WAIT_FOR_SHUTTLE, (*Load station is waiting for a shuttle to be present*)
		LOAD_LOADING, (*Load station is loading product onto a shuttle*)
		LOAD_DONE, (*Load station is done with the load process*)
		LOAD_ERROR (*Load station had an error*)
		);
	LoadStationFbTyp : 	STRUCT
		LoadTimerFb : TON;
	END_STRUCT;
END_TYPE
```

#### LocalFunctionVars.var
```iecst
VAR CONSTANT
	MAX_BATCH_SHUTTLE_COUNT : USINT := 2;
	MAX_BATCH_SHUTTLE_COUNT_ARRAY : USINT := MAX_BATCH_SHUTTLE_COUNT-1;
END_VAR
```

#### Variables.var
```iecst
VAR
	state : LoadStationStateEnum;
	LoadStationFbs : LoadStationFbTyp;
END_VAR
```

#### BatchProcess6DFb.st
```iecst
(* TODO: Add your comment here *)
FUNCTION_BLOCK BatchProcess6DFb
	CASE Internal.State OF
		BATCH_OFF://******************************************************************************** Batch FB disabled
			IF Enable THEN
				Internal.State := BATCH_INIT;
			END_IF
		BATCH_INIT://******************************************************************************** Batch FB Initialization state
			Internal.Fbs.MoveInPlaneFb.Controller := ADR(Controller);
			ReadyForShuttle := TRUE;

			Internal.State := BATCH_WAIT_SHUTTLE;
		BATCH_WAIT_SHUTTLE://******************************************************************************** Batch FB Waiting for a shuttle to arrive
			IF ProcessShuttle THEN
				Internal.currentShuttleCount := Internal.currentShuttleCount + 1;
				ReadyForShuttle := FALSE;
				IF ShId = 0 THEN
					Error := TRUE;
					Internal.State := BATCH_ERROR;
				ELSE
					ProcessShuttle := FALSE;

					ShuttleIds[Internal.currentShuttleCount - 1] := ShId;
					Internal.Fbs.MoveInPlaneFb.ShuttleID := ShId;
					Internal.Fbs.MoveInPlaneFb.Velocity := 1.0;
					Internal.Fbs.MoveInPlaneFb.Acceleration := 10.0;
					Internal.Fbs.MoveInPlaneFb.PositionX := Positions[Internal.currentShuttleCount - 1].X;
					Internal.Fbs.MoveInPlaneFb.PositionY := Positions[Internal.currentShuttleCount - 1].Y;
					Internal.Fbs.MoveInPlaneFb.Path := mcACP6D_PATH_X_THEN_Y;

					Internal.Fbs.MoveInPlaneFb.Execute := TRUE;

					Internal.State := BATCH_MOVE_SHUTTLE;
				END_IF
			END_IF
		BATCH_MOVE_SHUTTLE://******************************************************************************** Batch FB Move Shuttle State
			IF Internal.Fbs.MoveInPlaneFb.Error THEN
				Error := TRUE;
				StatusID := Internal.Fbs.MoveInPlaneFb.ErrorID;
				Internal.State := BATCH_ERROR;
			ELSIF (Internal.currentShuttleCount <> MAX_BATCH_SHUTTLE_COUNT AND Internal.Fbs.MoveInPlaneFb.Acknowledge) THEN
				Internal.Fbs.MoveInPlaneFb.Execute := FALSE;

				//The command has been added to the buffer but we're stil need more shuttles
				ReadyForShuttle := TRUE;

				Internal.State := BATCH_WAIT_SHUTTLE;
			ELSIF Internal.Fbs.MoveInPlaneFb.Done THEN
				//We are now going to start preforming the actual operation
				Internal.Fbs.MoveInPlaneFb.Execute := FALSE;
				Processsing := TRUE;
				Internal.Fbs.WaitTimer.IN := TRUE;
				Internal.Fbs.WaitTimer.PT := ProcessingTime;

				Internal.State := BATCH_PREFORM_OPERATION;
			END_IF
		BATCH_PREFORM_OPERATION://******************************************************************************** Batch FB Preforming the operation
			IF Internal.Fbs.WaitTimer.Q THEN
				Internal.Fbs.WaitTimer.IN := FALSE;

				Processsing := FALSE;
				BatchComplete := TRUE;

				Internal.State := BATCH_DONE;

			END_IF
		BATCH_DONE://******************************************************************************** Batch FB Done state
			IF Reset THEN
				Internal.State := BATCH_RESET;
			END_IF
		BATCH_RESET://******************************************************************************** Batch Reset all data state
			Reset := FALSE;

			BatchComplete := FALSE;
			Processsing := FALSE;
			ReadyForShuttle := FALSE;
			Error := FALSE;
			StatusID := FALSE;
			brsmemset(ADR(ShuttleIds),0,SIZEOF(ShuttleIds));

			Internal.currentShuttleCount := 0;

			Internal.Fbs.MoveInPlaneFb.Execute := FALSE;
			Internal.Fbs.WaitTimer.IN := FALSE;

			IF Enable THEN
				Internal.State := BATCH_INIT;
			ELSE
				Internal.State := BATCH_OFF;
			END_IF
		BATCH_ERROR://******************************************************************************** Batch FB Error state
			IF Reset THEN
				Internal.State := BATCH_RESET;
			END_IF
	END_CASE;
	Internal.Fbs.MoveInPlaneFb();
	Internal.Fbs.WaitTimer();
END_FUNCTION_BLOCK
```

#### Cyclic.st
```iecst
PROGRAM _CYCLIC
	CASE state OF
		LOAD_OFF: //********************************************************************************Load station is currently disabled
			IF gLoadStationIf.Cmd.Enable THEN
				state := LOAD_INIT;
			END_IF
		LOAD_INIT: //********************************************************************************Load station is initalizing
			gLoadStationIf.Status.ReadyForNewShuttle := TRUE;
			gLoadStationIf.Status.Enabled := TRUE;
			state := LOAD_WAIT_FOR_SHUTTLE;
		LOAD_WAIT_FOR_SHUTTLE: //********************************************************************************Load station is waiting for a shuttle to be present
			IF NOT gLoadStationIf.Cmd.Enable THEN
				gLoadStationIf.Status.ReadyForNewShuttle := FALSE;
				gLoadStationIf.Status.Enabled := FALSE;
				state := LOAD_OFF;
			ELSIF gLoadStationIf.Par.ShuttleIdx <> STATION_IS_EMPTY AND gLoadStationIf.Cmd.Process THEN
				gLoadStationIf.Status.ReadyForNewShuttle := FALSE;
				gLoadStationIf.Status.Processing := TRUE;

				LoadStationFbs.LoadTimerFb.IN := TRUE;
				LoadStationFbs.LoadTimerFb.PT := gLoadStationIf.Par.WaitTime;

				state := LOAD_LOADING;
			END_IF
		LOAD_LOADING: //********************************************************************************Load station is loading product onto a shuttle
			IF LoadStationFbs.LoadTimerFb.Q THEN
				LoadStationFbs.LoadTimerFb.IN := FALSE;

				gLoadStationIf.Status.Processing := FALSE;
				gShuttleIf[gLoadStationIf.Par.ShuttleIdx].Cmd.NextStep := TRUE;
				gLoadStationIf.Status.Done := TRUE;

				state := LOAD_DONE;
			END_IF
		LOAD_DONE: //********************************************************************************Load station is done with the load process
			IF NOT gLoadStationIf.Cmd.Enable THEN
				gLoadStationIf.Status.Done := FALSE;
				gLoadStationIf.Status.Enabled := FALSE;
				gLoadStationIf.Status.ReadyForNewShuttle := FALSE;
				state := LOAD_OFF;
			ELSIF NOT gLoadStationIf.Cmd.Process THEN
				gLoadStationIf.Par.ShuttleIdx := STATION_IS_EMPTY;
				gLoadStationIf.Status.Done := FALSE;
				gLoadStationIf.Status.ReadyForNewShuttle := FALSE;
				gLoadStationIf.Status.ReadyForNewShuttle := TRUE;

				state := LOAD_WAIT_FOR_SHUTTLE;
			END_IF

		LOAD_ERROR: //********************************************************************************Load station had an error
			IF gLoadStationIf.Cmd.Reset THEN
				gLoadStationIf.Cmd.Reset := FALSE;

				gLoadStationIf.Status.Done := FALSE;
				gLoadStationIf.Status.Enabled := FALSE;
				gLoadStationIf.Status.Error := FALSE;
				gLoadStationIf.Status.Processing := FALSE;
				gLoadStationIf.Status.ReadyForNewShuttle := FALSE;

				gLoadStationIf.Par.ShuttleIdx := STATION_IS_EMPTY;
				IF gLoadStationIf.Cmd.Enable THEN
					state := LOAD_INIT;
				ELSE
					state := LOAD_OFF;
				END_IF
			END_IF
	END_CASE;

	 LoadStationFbs.LoadTimerFb();
END_PROGRAM
```

#### Init.st
```iecst
PROGRAM _INIT
	gLoadStationIf.Par.ShuttleIdx := STATION_IS_EMPTY;
	//Define station configuration values
	gLoadStationIf.Cfg.StationPos.X := 0.060;
	gLoadStationIf.Cfg.StationPos.Y := 0.180;

	gLoadStationIf.Par.WaitTime := T#2s;

END_PROGRAM
```

### Program Logical/Source/ProcessStations/UnloadStation (IEC)

#### Types.typ
```iecst
TYPE
	UnloadStationStateEnum :
		(
		UNLOAD_OFF, (*Unload station is currently disabled*)
		UNLOAD_INIT, (*Unload station is initalizing*)
		UNLOAD_WAIT_FOR_SHUTTLE, (*Unload station is waiting for a shuttle to be present*)
		UNLOAD_UNLOADING, (*Unload station is loading product onto a shuttle*)
		UNLOAD_DONE, (*Unload station is done with the load process*)
		UNLOAD_ERROR (*Unload station had an error*)
		);
	UnloadStationFbTyp : 	STRUCT
		UnloadTimerFb : TON;
	END_STRUCT;
END_TYPE
```

#### LocalFunctionVars.var
```iecst
VAR CONSTANT
	MAX_BATCH_SHUTTLE_COUNT : USINT := 4;
	MAX_BATCH_SHUTTLE_COUNT_ARRAY : USINT := MAX_BATCH_SHUTTLE_COUNT-1;
END_VAR
```

#### Variables.var
```iecst
VAR
	state : UnloadStationStateEnum;
	UnloadStationFbs : UnloadStationFbTyp;
END_VAR
```

#### Cyclic.st
```iecst
PROGRAM _CYCLIC
	CASE state OF
		UNLOAD_OFF: //********************************************************************************Unload station is currently disabled
			IF gUnloadStationIf.Cmd.Enable THEN
				state := UNLOAD_INIT;
			END_IF
		UNLOAD_INIT: //********************************************************************************Unload station is initalizing
			gUnloadStationIf.Status.ReadyForNewShuttle := TRUE;
			gUnloadStationIf.Status.Enabled := TRUE;
			state := UNLOAD_WAIT_FOR_SHUTTLE;
		UNLOAD_WAIT_FOR_SHUTTLE: //********************************************************************************Unload station is waiting for a shuttle to be present
			IF NOT gUnloadStationIf.Cmd.Enable THEN
				gUnloadStationIf.Status.ReadyForNewShuttle := FALSE;
				gUnloadStationIf.Status.Enabled := FALSE;
				state := UNLOAD_OFF;
			ELSIF gUnloadStationIf.Par.ShuttleIdx <> STATION_IS_EMPTY AND gUnloadStationIf.Cmd.Process THEN
				gUnloadStationIf.Status.ReadyForNewShuttle := FALSE;
				gUnloadStationIf.Status.Processing := TRUE;

				UnloadStationFbs.UnloadTimerFb.IN := TRUE;
				UnloadStationFbs.UnloadTimerFb.PT := gUnloadStationIf.Par.WaitTime;

				state := UNLOAD_UNLOADING;
			END_IF
		UNLOAD_UNLOADING: //********************************************************************************Unload station is unloading product off a shuttle
			IF UnloadStationFbs.UnloadTimerFb.Q THEN
				UnloadStationFbs.UnloadTimerFb.IN := FALSE;

				gUnloadStationIf.Status.Processing := FALSE;
				gShuttleIf[gUnloadStationIf.Par.ShuttleIdx].Cmd.NextStep := TRUE;
				gUnloadStationIf.Status.Done := TRUE;

				state := UNLOAD_DONE;
			END_IF
		UNLOAD_DONE: //********************************************************************************Unload station is done with the unload process
			IF NOT gUnloadStationIf.Cmd.Enable THEN
				gUnloadStationIf.Status.Done := FALSE;
				gUnloadStationIf.Status.Enabled := FALSE;
				gUnloadStationIf.Status.ReadyForNewShuttle := FALSE;
				state := UNLOAD_OFF;
			ELSIF NOT gUnloadStationIf.Cmd.Process THEN
				gUnloadStationIf.Par.ShuttleIdx := STATION_IS_EMPTY;
				gUnloadStationIf.Status.ReadyForNewShuttle := FALSE;
				gUnloadStationIf.Status.ReadyForNewShuttle := TRUE;

				state := UNLOAD_WAIT_FOR_SHUTTLE;
			END_IF

		UNLOAD_ERROR: //********************************************************************************Unload station had an error
			IF gUnloadStationIf.Cmd.Reset THEN
				gUnloadStationIf.Cmd.Reset := FALSE;

				gUnloadStationIf.Status.Done := FALSE;
				gUnloadStationIf.Status.Enabled := FALSE;
				gUnloadStationIf.Status.Error := FALSE;
				gUnloadStationIf.Status.Processing := FALSE;
				gUnloadStationIf.Status.ReadyForNewShuttle := FALSE;

				gUnloadStationIf.Par.ShuttleIdx := STATION_IS_EMPTY;
				IF gUnloadStationIf.Cmd.Enable THEN
					state := UNLOAD_INIT;
				ELSE
					state := UNLOAD_OFF;
				END_IF
			END_IF
	END_CASE;

	UnloadStationFbs.UnloadTimerFb();
END_PROGRAM
```

#### Init.st
```iecst
PROGRAM _INIT
	gUnloadStationIf.Par.ShuttleIdx := STATION_IS_EMPTY;
	//Define station configuration values
	gUnloadStationIf.Cfg.StationPos.X := 0.060;
	gUnloadStationIf.Cfg.StationPos.Y := 0.3;

	gUnloadStationIf.Par.WaitTime := T#2s;
END_PROGRAM
```

### Program Logical/Source/ProcessStations/DoseStation (IEC)

#### Types.typ
```iecst
TYPE
	DoseStationStateEnum :
		(
		DOSE_OFF, (*Dose station is currently disabled*)
		DOSE_INIT, (*Dose station is initalizing*)
		DOSE_WAIT_FOR_SHUTTLE, (*Dose station is waiting for a shuttle to be present*)
		DOSE_INDEX_SHUTTLE, (*Dose station is indexing to the next dosing position*)
		DOSE_DOSING, (*Dose station is preforming the dosing process*)
		DOSE_DONE, (*Dose station is done with the dosing process*)
		DOSE_ERROR (*Dose station had an error*)
		);
	DoseStationFbTyp : 	STRUCT
		DoseMoveFb : MC_BR_MoveInPlane_Acp6D;
		WaitTimer : TON;
	END_STRUCT;
END_TYPE
```

#### Variables.var
```iecst
VAR
	state : DoseStationStateEnum;
	pDoseIf : REFERENCE TO DoseStationIfTyp;
	DoseStationFbs : DoseStationFbTyp;
	currentRow : USINT; (*Current row the process is on for indexing through the dosing process*)
	taskName : STRING[80];
	tmp : WSTRING[80];
	msgType : WSTRING[80];
	msgMsg : WSTRING[80];
END_VAR
```

#### Cyclic.st
```iecst
PROGRAM _CYCLIC
	CASE state OF
		DOSE_OFF: //********************************************************************************Dose station is currently disabled
			IF pDoseIf.Cmd.Enable THEN
				state := DOSE_INIT;
			END_IF
		DOSE_INIT: //********************************************************************************Dose station is initalizing
			pDoseIf.Status.ReadyForNewShuttle := TRUE;
			pDoseIf.Status.Enabled := TRUE;
			state := DOSE_WAIT_FOR_SHUTTLE;
		DOSE_WAIT_FOR_SHUTTLE: //********************************************************************************Dose station is waiting for a shuttle to be present
			IF NOT pDoseIf.Cmd.Enable THEN
				pDoseIf.Status.ReadyForNewShuttle := FALSE;
				pDoseIf.Status.Enabled := FALSE;
				state := DOSE_OFF;
			ELSIF pDoseIf.Par.ShuttleIdx <> STATION_IS_EMPTY AND pDoseIf.Cmd.Process THEN
				pDoseIf.Status.ReadyForNewShuttle := FALSE;
				pDoseIf.Status.Processing := TRUE;

				DoseStationFbs.DoseMoveFb.Controller := ADR(gMcAcp6DController);
				DoseStationFbs.DoseMoveFb.ShuttleID := gShuttleIf[pDoseIf.Par.ShuttleIdx].Cfg.ShuttleId;
				DoseStationFbs.DoseMoveFb.Mode := mcACP6D_MOVE_RELATIVE;
				DoseStationFbs.DoseMoveFb.Path := mcACP6D_PATH_DIRECT;
				DoseStationFbs.DoseMoveFb.Velocity := pDoseIf.Par.Vel;
				DoseStationFbs.DoseMoveFb.EndVelocity := pDoseIf.Par.EndVel;
				DoseStationFbs.DoseMoveFb.Acceleration := pDoseIf.Par.Accel;
				DoseStationFbs.DoseMoveFb.PositionX := (pDoseIf.Par.FirstCavityPosition.DistX);
				DoseStationFbs.DoseMoveFb.PositionY := -(pDoseIf.Par.FirstCavityPosition.DistY); //Made negative as we're moving in negative Z
				DoseStationFbs.DoseMoveFb.Execute := TRUE;

//				msgType := "";
//				msgMsg := "";
//				tmp := STRING_TO_WSTRING(taskName);
//				brwcscat(ADR(msgType),ADR(tmp));
//				brwcscat(ADR(msgType),ADR(":FirstMove:Sh"));
//				tmp := USINT_TO_WSTRING(gShuttleIf[pDoseIf.Par.ShuttleIdx].Cfg.ShuttleId);
//				brwcscat(ADR(msgType),ADR(tmp));
//				tmp := "";
//				msgMsg := "X:";
//				tmp := REAL_TO_WSTRING(DoseStationFbs.DoseMoveFb.PositionX);
//				brwcscat(ADR(msgMsg),ADR(tmp));
//				brwcscat(ADR(msgMsg),ADR(" Y:"));
//				tmp := REAL_TO_WSTRING(DoseStationFbs.DoseMoveFb.PositionY);
//				brwcscat(ADR(msgMsg),ADR(tmp));
//				MpAuditCustomEvent(gAuditTrail,"DEBUG",msgType,msgMsg);

				state := DOSE_INDEX_SHUTTLE;
			END_IF
		DOSE_INDEX_SHUTTLE: //******************************************************************************** Dose station is indexing to the next dosing position
			IF DoseStationFbs.DoseMoveFb.Error THEN
				pDoseIf.Status.Error := TRUE;

				state := DOSE_ERROR;
			ELSIF DoseStationFbs.DoseMoveFb.Done THEN
				DoseStationFbs.DoseMoveFb.Execute:= FALSE;

				DoseStationFbs.WaitTimer.IN := TRUE;
				DoseStationFbs.WaitTimer.PT := pDoseIf.Par.WaitTime;

				state := DOSE_DOSING;
			END_IF
		DOSE_DOSING: //********************************************************************************Dose station is preforming the dosing process
			IF DoseStationFbs.WaitTimer.Q THEN
				DoseStationFbs.WaitTimer.IN := FALSE;
				gProcessInfoIf.Par.CurrentPowderCount := gProcessInfoIf.Par.CurrentPowderCount + 1;
				currentRow := currentRow + 1;
				IF currentRow > (pDoseIf.Par.NumRowsOfCavities-1) THEN
					gShuttleIf[pDoseIf.Par.ShuttleIdx].Cmd.NextStep := TRUE;
					pDoseIf.Status.Done := TRUE;
					pDoseIf.Status.Processing := FALSE;

					state := DOSE_DONE;
				ELSE
					DoseStationFbs.DoseMoveFb.Controller := ADR(gMcAcp6DController);
					DoseStationFbs.DoseMoveFb.ShuttleID := gShuttleIf[pDoseIf.Par.ShuttleIdx].Cfg.ShuttleId;
					DoseStationFbs.DoseMoveFb.Mode := mcACP6D_MOVE_RELATIVE;
					DoseStationFbs.DoseMoveFb.Path := mcACP6D_PATH_DIRECT;
					DoseStationFbs.DoseMoveFb.Velocity := pDoseIf.Par.Vel;
					DoseStationFbs.DoseMoveFb.EndVelocity := pDoseIf.Par.EndVel;
					DoseStationFbs.DoseMoveFb.Acceleration := pDoseIf.Par.Accel;
					DoseStationFbs.DoseMoveFb.PositionX := (pDoseIf.Par.SpaceBetweenCavities.DistX);
					DoseStationFbs.DoseMoveFb.PositionY := -(pDoseIf.Par.SpaceBetweenCavities.DistY); //Made negative as we're moving in negative Z
					DoseStationFbs.DoseMoveFb.Execute := TRUE;

					state := DOSE_INDEX_SHUTTLE;
				END_IF
			END_IF
		DOSE_DONE: //********************************************************************************Dose station is done with the load process
			IF NOT pDoseIf.Cmd.Enable THEN
				pDoseIf.Status.Enabled := FALSE;
				pDoseIf.Status.ReadyForNewShuttle := FALSE;
				currentRow := 0;

				state := DOSE_OFF;
			ELSIF NOT pDoseIf.Cmd.Process THEN
				pDoseIf.Status.Done := FALSE;
				currentRow := 0;

				pDoseIf.Par.ShuttleIdx := STATION_IS_EMPTY;
				pDoseIf.Status.ReadyForNewShuttle := FALSE;
				pDoseIf.Status.ReadyForNewShuttle := TRUE;

				state := DOSE_WAIT_FOR_SHUTTLE;
			END_IF
		DOSE_ERROR: //********************************************************************************Dose station had an error
			IF pDoseIf.Cmd.Reset THEN
				pDoseIf.Cmd.Reset := FALSE;

				pDoseIf.Par.ShuttleIdx := STATION_IS_EMPTY;

				currentRow := 0;

				pDoseIf.Status.Done := FALSE;
				pDoseIf.Status.Error := FALSE;
				pDoseIf.Status.Processing := FALSE;
				pDoseIf.Status.ReadyForNewShuttle := FALSE;
				pDoseIf.Status.Enabled := FALSE;

				DoseStationFbs.DoseMoveFb.Execute := FALSE;
				DoseStationFbs.WaitTimer.IN := FALSE;

				IF pDoseIf.Cmd.Enable THEN
					state := DOSE_INIT;
				ELSE
					state := DOSE_OFF;
				END_IF
			END_IF
	END_CASE;

	DoseStationFbs.DoseMoveFb();
	DoseStationFbs.WaitTimer();
END_PROGRAM
```

#### Init.st
```iecst
PROGRAM _INIT
	ST_name(0,ADR(taskName),0);

	IF taskName = 'DoseSt1' THEN
		pDoseIf ACCESS ADR(gDoseStationsIf[0]);
	ELSIF taskName = 'DoseSt2' THEN
		pDoseIf ACCESS ADR(gDoseStationsIf[1]);
	END_IF

	gDoseStationsIf[0].Cfg.StationPos.X := 0.3;
	gDoseStationsIf[0].Cfg.StationPos.Y := 0.66;

	gDoseStationsIf[1].Cfg.StationPos.X := 0.66;
	gDoseStationsIf[1].Cfg.StationPos.Y := 0.66;

	pDoseIf.Par.ShuttleIdx := STATION_IS_EMPTY;
	pDoseIf.Par.Accel := 0.3;
	pDoseIf.Par.Vel := 0.508;
	pDoseIf.Par.EndVel := 0.0;
	pDoseIf.Par.FirstCavityPosition.DistY := 0.03;
	pDoseIf.Par.FirstCavityPosition.DistX := 0.0;

	pDoseIf.Par.SpaceBetweenCavities.DistY := 0.03;
	pDoseIf.Par.SpaceBetweenCavities.DistX := 0;
	pDoseIf.Par.NumRowsOfCavities := 3;
	pDoseIf.Par.WaitTime := T#2s;
END_PROGRAM
```

### Program Logical/Source/ProcessStations/PrintStation (IEC)

#### Types.typ
```iecst
TYPE
	PrintStationStateEnum :
		(
		PRINT_OFF, (*Print station is currently disabled*)
		PRINT_INIT, (*Print station is initalizing*)
		PRINT_WAIT_FOR_SHUTTLE, (*Print station is waiting for a shuttle to be present*)
		PRINT_PRINTING, (*Print station is moving through the print process*)
		PRINT_DONE, (*Print station is done with the print process*)
		PRINT_ERROR (*Print station had an error*)
		);
	PrintStationFbTyp : 	STRUCT
		PrintMoveFb : MC_BR_MoveInPlane_Acp6D;
	END_STRUCT;
END_TYPE
```

#### Variables.var
```iecst
VAR
	state : PrintStationStateEnum;
	PrintStationFbs : PrintStationFbTyp;
END_VAR
```

#### Cyclic.st
```iecst
PROGRAM _CYCLIC
	CASE state OF
		PRINT_OFF: //********************************************************************************Print station is currently disabled
			IF gPrintStationIf.Cmd.Enable THEN
				state := PRINT_INIT;
			END_IF
		PRINT_INIT: //********************************************************************************Print station is initalizing
			gPrintStationIf.Status.ReadyForNewShuttle := TRUE;
			gPrintStationIf.Status.Enabled := TRUE;
			state := PRINT_WAIT_FOR_SHUTTLE;
		PRINT_WAIT_FOR_SHUTTLE: //********************************************************************************Print station is waiting for a shuttle to be present
			IF NOT gPrintStationIf.Cmd.Enable THEN
				gPrintStationIf.Status.ReadyForNewShuttle := FALSE;
				gPrintStationIf.Status.Enabled := FALSE;
				state := PRINT_OFF;
			ELSIF gPrintStationIf.Par.ShuttleIdx <> STATION_IS_EMPTY AND gPrintStationIf.Cmd.Process THEN
				gPrintStationIf.Status.ReadyForNewShuttle := FALSE;
				gPrintStationIf.Status.Processing := TRUE;

				PrintStationFbs.PrintMoveFb.Controller := ADR(gMcAcp6DController);
				PrintStationFbs.PrintMoveFb.ShuttleID := gShuttleIf[gPrintStationIf.Par.ShuttleIdx].Cfg.ShuttleId;
				PrintStationFbs.PrintMoveFb.Mode := mcACP6D_MOVE_RELATIVE;
				PrintStationFbs.PrintMoveFb.Path := mcACP6D_PATH_DIRECT;
				PrintStationFbs.PrintMoveFb.Velocity := gPrintStationIf.Par.PrintVel;
				PrintStationFbs.PrintMoveFb.EndVelocity := gPrintStationIf.Par.PrintAccel;
				PrintStationFbs.PrintMoveFb.Acceleration := gPrintStationIf.Par.PrintAccel;
				PrintStationFbs.PrintMoveFb.PositionX := gPrintStationIf.Par.PrintDistanceX;
				PrintStationFbs.PrintMoveFb.PositionY := gPrintStationIf.Par.PrintDistanceY;
				PrintStationFbs.PrintMoveFb.Execute := TRUE;

				state := PRINT_PRINTING;
			END_IF
		PRINT_PRINTING: //********************************************************************************Print station is loading product onto a shuttle
			IF PrintStationFbs.PrintMoveFb.Error THEN
				gPrintStationIf.Status.Error := TRUE;

				state := PRINT_ERROR;
			ELSIF PrintStationFbs.PrintMoveFb.Done THEN
				PrintStationFbs.PrintMoveFb.Execute:= FALSE;

				gPrintStationIf.Status.Processing := FALSE;
				gShuttleIf[gPrintStationIf.Par.ShuttleIdx].Cmd.NextStep := TRUE; //Tell the shuttle we've finished the process and it's okay to move on to the next step
				gPrintStationIf.Status.Done := TRUE;

				state := PRINT_DONE;
			END_IF
		PRINT_DONE: //********************************************************************************Print station is done with the load process
			IF NOT gPrintStationIf.Cmd.Enable THEN
				gPrintStationIf.Status.Enabled := FALSE;
				gPrintStationIf.Status.ReadyForNewShuttle := FALSE;
				state := PRINT_OFF;
			ELSIF NOT gPrintStationIf.Cmd.Process THEN
				gPrintStationIf.Status.Done := FALSE;

				gPrintStationIf.Par.ShuttleIdx := STATION_IS_EMPTY;
				gPrintStationIf.Status.ReadyForNewShuttle := FALSE;
				gPrintStationIf.Status.ReadyForNewShuttle := TRUE;

				state := PRINT_WAIT_FOR_SHUTTLE;
			END_IF
		PRINT_ERROR: //********************************************************************************Print station had an error
			IF gPrintStationIf.Cmd.Reset THEN
				gPrintStationIf.Cmd.Reset := FALSE;

				gPrintStationIf.Par.ShuttleIdx := STATION_IS_EMPTY;

				gPrintStationIf.Status.Done := FALSE;
				gPrintStationIf.Status.Error := FALSE;
				gPrintStationIf.Status.Processing := FALSE;
				gPrintStationIf.Status.ReadyForNewShuttle := FALSE;
				gPrintStationIf.Status.Enabled := FALSE;

				PrintStationFbs.PrintMoveFb.Execute := FALSE;

				IF gPrintStationIf.Cmd.Enable THEN
					state := PRINT_INIT;
				ELSE
					state := PRINT_OFF;
				END_IF
			END_IF
	END_CASE;

	PrintStationFbs.PrintMoveFb();
END_PROGRAM
```

#### Init.st
```iecst
PROGRAM _INIT
	gPrintStationIf.Par.ShuttleIdx := STATION_IS_EMPTY;
	//Define station configuration values
	gPrintStationIf.Cfg.StationPos.X := 0.30;
	gPrintStationIf.Cfg.StationPos.Y := 0.06;

	gPrintStationIf.Par.PrintAccel := 0.30;
	gPrintStationIf.Par.PrintVel := 0.2302; //8 in/s
	gPrintStationIf.Par.PrintEndVel :=  0.0;
	gPrintStationIf.Par.PrintDistanceX := 0.12;
	gPrintStationIf.Par.PrintDistanceY := 0;

END_PROGRAM
```

### Program Logical/Source/ProcessStations/TampStation (IEC)

#### Types.typ
```iecst
TYPE
	TampStationStateEnum :
		(
		TAMP_OFF, (*Tamp station is currently disabled*)
		TAMP_INIT, (*Tamp station is initalizing*)
		TAMP_WAIT_FOR_SHUTTLE, (*Tamp station is waiting for a shuttle to be present*)
		TAMP_ENTER_STATION, (*Tamp station is sending the shuttle to the tamp position*)
		TAMP_TAMP_RAISE, (*Tamp station is preforming the lift for the tamp process*)
		TAMP_TAMPING, (*Tamp station is waiting at the tamp height*)
		TAMP_TAMP_LOWER, (*Tamp station is performing the lower for the tamp process*)
		TAMP_EXIT_STATION, (*Tamps tation is sending the shuttle to the exit point*)
		TAMP_DONE, (*Tamp station is done with the dosing process*)
		TAMP_ERROR (*Tamp station had an error*)
		);
	TampStationFbTyp : 	STRUCT
		TampMoveFb : MC_BR_MoveInPlane_Acp6D;
		ShortAxisFb : MC_BR_MoveShortAxis_Acp6D;
		WaitTimer : TON;
	END_STRUCT;
END_TYPE
```

#### Variables.var
```iecst
VAR
	state : TampStationStateEnum;
	TampStationFbs : TampStationFbTyp;
END_VAR
```

#### Cyclic.st
```iecst
PROGRAM _CYCLIC
	CASE state OF
		TAMP_OFF: //********************************************************************************Tamp station is currently disabled
			IF gTampStationIf.Cmd.Enable THEN
				state := TAMP_INIT;
			END_IF
		TAMP_INIT: //********************************************************************************Tamp station is initalizing
			gTampStationIf.Status.ReadyForNewShuttle := TRUE;
			gTampStationIf.Status.Enabled := TRUE;
			state := TAMP_WAIT_FOR_SHUTTLE;
		TAMP_WAIT_FOR_SHUTTLE: //********************************************************************************Tamp station is waiting for a shuttle to be present
			IF NOT gTampStationIf.Cmd.Enable THEN
				gTampStationIf.Status.ReadyForNewShuttle := FALSE;
				gTampStationIf.Status.Enabled := FALSE;
				state := TAMP_OFF;
			ELSIF gTampStationIf.Par.ShuttleIdx <> STATION_IS_EMPTY AND gTampStationIf.Cmd.Process THEN
				gTampStationIf.Status.ReadyForNewShuttle := FALSE;
				gTampStationIf.Status.Processing := TRUE;

				TampStationFbs.TampMoveFb.Controller := ADR(gMcAcp6DController);
				TampStationFbs.TampMoveFb.ShuttleID := gShuttleIf[gTampStationIf.Par.ShuttleIdx].Cfg.ShuttleId;
				TampStationFbs.TampMoveFb.Mode := mcACP6D_MOVE_RELATIVE;
				TampStationFbs.TampMoveFb.Path := mcACP6D_PATH_DIRECT;
				TampStationFbs.TampMoveFb.Velocity := gTampStationIf.Par.Vel;
				TampStationFbs.TampMoveFb.EndVelocity := gTampStationIf.Par.EndVel;
				TampStationFbs.TampMoveFb.Acceleration := gTampStationIf.Par.Accel;
				TampStationFbs.TampMoveFb.PositionX := gTampStationIf.Par.EntranceMovement.DistX;
				TampStationFbs.TampMoveFb.PositionY := gTampStationIf.Par.EntranceMovement.DistY;
				TampStationFbs.TampMoveFb.Execute := TRUE;

				state := TAMP_ENTER_STATION;
			END_IF
		TAMP_ENTER_STATION: //******************************************************************************** Tamp station is sending the shuttle to the tamp position
			IF TampStationFbs.TampMoveFb.Error THEN
				gTampStationIf.Status.Error := TRUE;

				state := TAMP_ERROR;
			ELSIF TampStationFbs.TampMoveFb.Done THEN
				TampStationFbs.TampMoveFb.Execute:= FALSE;

				TampStationFbs.ShortAxisFb.Controller := ADR(gMcAcp6DController);
				TampStationFbs.ShortAxisFb.ShuttleID := gShuttleIf[gTampStationIf.Par.ShuttleIdx].Cfg.ShuttleId;
				TampStationFbs.ShortAxisFb.Mode := mcACP6D_MOVE_RELATIVE;
				TampStationFbs.ShortAxisFb.PositionZ := gTampStationIf.Par.TampHeight;
				TampStationFbs.ShortAxisFb.VelocityZ := gTampStationIf.Par.Vel;
				TampStationFbs.ShortAxisFb.Execute := TRUE;

				state := TAMP_TAMP_RAISE;
			END_IF
		TAMP_TAMP_RAISE: //******************************************************************************** Tamp station is raising to the tamp height
			IF TampStationFbs.ShortAxisFb.Error THEN
				gTampStationIf.Status.Error := TRUE;

				state := TAMP_ERROR;
			ELSIF TampStationFbs.ShortAxisFb.Done THEN
				TampStationFbs.ShortAxisFb.Execute:= FALSE;

				TampStationFbs.WaitTimer.IN := TRUE;
				TampStationFbs.WaitTimer.PT := gTampStationIf.Par.WaitTime;

				state := TAMP_TAMPING;
			END_IF

		TAMP_TAMPING: //********************************************************************************Tamp station is preforming the tamping process
			IF TampStationFbs.WaitTimer.Q THEN
				TampStationFbs.WaitTimer.IN := FALSE;

				TampStationFbs.ShortAxisFb.Controller := ADR(gMcAcp6DController);
				TampStationFbs.ShortAxisFb.ShuttleID := gShuttleIf[gTampStationIf.Par.ShuttleIdx].Cfg.ShuttleId;
				TampStationFbs.ShortAxisFb.Mode := mcACP6D_MOVE_RELATIVE;
				TampStationFbs.ShortAxisFb.PositionZ := -gTampStationIf.Par.TampHeight;
				TampStationFbs.ShortAxisFb.VelocityZ := gTampStationIf.Par.Vel;
				TampStationFbs.ShortAxisFb.Execute := TRUE;

				state := TAMP_TAMP_LOWER;
			END_IF
		TAMP_TAMP_LOWER: //******************************************************************************** Tamp station is raising to the tamp height
			IF TampStationFbs.ShortAxisFb.Error THEN
				gTampStationIf.Status.Error := TRUE;

				state := TAMP_ERROR;
			ELSIF TampStationFbs.ShortAxisFb.Done THEN
				TampStationFbs.ShortAxisFb.Execute:= FALSE;

				TampStationFbs.TampMoveFb.Controller := ADR(gMcAcp6DController);
				TampStationFbs.TampMoveFb.ShuttleID := gShuttleIf[gTampStationIf.Par.ShuttleIdx].Cfg.ShuttleId;
				TampStationFbs.TampMoveFb.Mode := mcACP6D_MOVE_RELATIVE;
				TampStationFbs.TampMoveFb.Path := mcACP6D_PATH_Y_THEN_X;
				TampStationFbs.TampMoveFb.Velocity := gTampStationIf.Par.Vel;
				TampStationFbs.TampMoveFb.EndVelocity := gTampStationIf.Par.EndVel;
				TampStationFbs.TampMoveFb.Acceleration := gTampStationIf.Par.Accel;
				TampStationFbs.TampMoveFb.PositionX := gTampStationIf.Par.ExitMovement.DistX;
				TampStationFbs.TampMoveFb.PositionY := gTampStationIf.Par.ExitMovement.DistY;
				TampStationFbs.TampMoveFb.Execute := TRUE;

				state := TAMP_EXIT_STATION;
			END_IF
		TAMP_EXIT_STATION: //******************************************************************************** Tamp station is sending the shuttle to the exit position
			IF TampStationFbs.TampMoveFb.Error THEN
				gTampStationIf.Status.Error := TRUE;

				state := TAMP_ERROR;
			ELSIF TampStationFbs.TampMoveFb.Done THEN
				TampStationFbs.TampMoveFb.Execute:= FALSE;

				gTampStationIf.Status.Done := TRUE;
				gTampStationIf.Status.Processing := FALSE;
				gShuttleIf[gTampStationIf.Par.ShuttleIdx].Cmd.NextStep := TRUE;

				state := TAMP_DONE;
			END_IF
		TAMP_DONE: //********************************************************************************Tamp station is done with the load process
			IF NOT gTampStationIf.Cmd.Enable THEN
				gTampStationIf.Status.Enabled := FALSE;
				gTampStationIf.Status.ReadyForNewShuttle := FALSE;

				state := TAMP_OFF;
			ELSIF NOT gTampStationIf.Cmd.Process THEN
				gTampStationIf.Status.Done := FALSE;

				gTampStationIf.Par.ShuttleIdx := STATION_IS_EMPTY;
				gTampStationIf.Status.ReadyForNewShuttle := FALSE;
				gTampStationIf.Status.ReadyForNewShuttle := TRUE;

				state := TAMP_WAIT_FOR_SHUTTLE;
			END_IF
		TAMP_ERROR: //********************************************************************************Tamp station had an error
			IF gTampStationIf.Cmd.Reset THEN
				gTampStationIf.Cmd.Reset := FALSE;

				gTampStationIf.Par.ShuttleIdx := STATION_IS_EMPTY;

				gTampStationIf.Status.Done := FALSE;
				gTampStationIf.Status.Error := FALSE;
				gTampStationIf.Status.Processing := FALSE;
				gTampStationIf.Status.ReadyForNewShuttle := FALSE;
				gTampStationIf.Status.Enabled := FALSE;

				TampStationFbs.TampMoveFb.Execute := FALSE;
				TampStationFbs.ShortAxisFb.Execute := FALSE;
				TampStationFbs.WaitTimer.IN := FALSE;

				IF gTampStationIf.Cmd.Enable THEN
					state := TAMP_INIT;
				ELSE
					state := TAMP_OFF;
				END_IF
			END_IF
	END_CASE;

	TampStationFbs.TampMoveFb();
	TampStationFbs.ShortAxisFb();
	TampStationFbs.WaitTimer();
END_PROGRAM
```

#### Init.st
```iecst
PROGRAM _INIT
	gTampStationIf.Par.ShuttleIdx := STATION_IS_EMPTY;
	//Define station configuration values
	gTampStationIf.Cfg.StationPos.X := 0.660;
	gTampStationIf.Cfg.StationPos.Y := 0.06;

	gTampStationIf.Par.Accel := 0.30;
	gTampStationIf.Par.Vel := 0.508;
	gTampStationIf.Par.EndVel := 0;
	gTampStationIf.Par.EntranceMovement.DistX := 0.18;
	gTampStationIf.Par.EntranceMovement.DistY := 0.06;
	gTampStationIf.Par.TampHeight := 0.002;
	gTampStationIf.Par.ExitMovement.DistX := -0.18;
	gTampStationIf.Par.ExitMovement.DistY := 0.06;
	gTampStationIf.Par.WaitTime := T#100ms;

END_PROGRAM
```

### Program Logical/Source/ProcessStations/BufferArea

#### Types.typ
```iecst
TYPE
	BufferAreaStatesEnum :
		(
		BUFFER_OFF, (*Buffer station is currently disabled*)
		BUFFER_INIT, (*Buffer station is initalizing*)
		BUFFER_WAIT_FOR_SHUTTLE, (*Buffer station is waiting for a shuttle to be requested to be added*)
		BUFFER_ADDING_SHUTTLE, (*Buffer station is adding a shuttle to the buffer*)
		BUFFER_CALL_OFF_SHUTTLES, (*Buffer station is calling off shuttles to be removed from the buffer area*)
		BUFFER_DONE, (*Buffer station is done with the process*)
		BUFFER_ERROR (*Buffer station had an error*)
		);
END_TYPE
```

#### Variables.var
```iecst
VAR
	state : BufferAreaStatesEnum;
	bufferArea : BufferListTyp;
	returnVal : SINT;
	stationPars : BufferAreaParsTyp;
	i : INT;
	serveShuttleId : USINT;
	shId : SINT;
END_VAR
```

#### Cyclic.st
```iecst
PROGRAM _CYCLIC
	IF NOT gBufferAreaIf.Cmd.LocalOverride THEN
		stationPars := gSysPars.BufferArea;
	END_IF

	CASE state OF
		BUFFER_OFF: //********************************************************************************Buffer station is currently disabled
			IF gBufferAreaIf.Cmd.Enable THEN
				state := BUFFER_INIT;
			END_IF
		BUFFER_INIT: //********************************************************************************Buffer station is initalizing
			gBufferAreaIf.Sts.ReadyForNewShuttle := TRUE;
			gBufferAreaIf.Sts.Enabled := TRUE;
			state := BUFFER_WAIT_FOR_SHUTTLE;
		BUFFER_WAIT_FOR_SHUTTLE: //********************************************************************************Buffer station is waiting for a shuttle to be requested to be added
			IF NOT gBufferAreaIf.Cmd.Enable THEN
				gBufferAreaIf.Sts.ReadyForNewShuttle := FALSE;
				gBufferAreaIf.Sts.Enabled := FALSE;
				blResetList(ADR(bufferArea));

				state := BUFFER_OFF;
			ELSIF gBufferAreaIf.Par.ShuttleIdx <> STATION_IS_EMPTY AND gBufferAreaIf.Cmd.Process THEN
				gBufferAreaIf.Sts.ReadyForNewShuttle := FALSE;
				gBufferAreaIf.Sts.Processing := TRUE;

				state := BUFFER_ADDING_SHUTTLE;
			END_IF
		BUFFER_ADDING_SHUTTLE: //********************************************************************************Buffer station is adding a shuttle to the buffer
			returnVal := blAddItem(ADR(bufferArea),gBufferAreaIf.Par.ShuttleIdx);
			IF returnVal <> 0 THEN
				gBufferAreaIf.Sts.Error := TRUE;
				state := BUFFER_ERROR;
			ELSE
				gBufferAreaIf.Sts.Processing := FALSE;

				IF bufferArea.CurrentLength >= stationPars.MinBufferSize THEN
					state := BUFFER_CALL_OFF_SHUTTLES;
				ELSE
					gBufferAreaIf.Par.ShuttleIdx := STATION_IS_EMPTY;
					gBufferAreaIf.Sts.ReadyForNewShuttle := TRUE;

					state := BUFFER_WAIT_FOR_SHUTTLE;
				END_IF
			END_IF//********************************************************************************Buffer station is calling off shuttles to be removed from the buffer area
		BUFFER_CALL_OFF_SHUTTLES:
			//This is a little dangerous of a process
			(*
				Get a random shuttle number from 1 to the current length
				Remove that ID from the list to get the value at that index
				Use that value as the index for the gShuttle interface to command off the buffer
			*)
			WHILE bufferArea.CurrentLength > stationPars.MinBufferSize - 4 DO
				serveShuttleId := DINT_TO_USINT(RandValueDINT(1,bufferArea.CurrentLength));
				shId := blRemoveItem(ADR(bufferArea),serveShuttleId);
				gShuttleIf[SINT_TO_USINT(shId)].Cmd.NextStep := TRUE;

			END_WHILE;
			gBufferAreaIf.Par.ShuttleIdx := STATION_IS_EMPTY;
			gBufferAreaIf.Sts.ReadyForNewShuttle := TRUE;

			state := BUFFER_WAIT_FOR_SHUTTLE;
		BUFFER_DONE: //********************************************************************************Buffer station is done with the process

			IF NOT gBufferAreaIf.Cmd.Enable THEN
				gBufferAreaIf.Sts.Done := FALSE;
				gBufferAreaIf.Sts.Enabled := FALSE;
				gBufferAreaIf.Sts.ReadyForNewShuttle := FALSE;
				blResetList(ADR(bufferArea));
				state := BUFFER_OFF;
			ELSIF NOT gBufferAreaIf.Cmd.Process THEN
				gBufferAreaIf.Par.ShuttleIdx := STATION_IS_EMPTY;
				gBufferAreaIf.Sts.Done := FALSE;
				gBufferAreaIf.Sts.ReadyForNewShuttle := TRUE;

				state := BUFFER_WAIT_FOR_SHUTTLE;
			END_IF

		BUFFER_ERROR: //********************************************************************************Load station had an error
			IF gBufferAreaIf.Cmd.Reset THEN
				gBufferAreaIf.Cmd.Reset := FALSE;

				blResetList(ADR(bufferArea));

				gBufferAreaIf.Sts.Done := FALSE;
				gBufferAreaIf.Sts.Enabled := FALSE;
				gBufferAreaIf.Sts.Error := FALSE;
				gBufferAreaIf.Sts.Processing := FALSE;
				gBufferAreaIf.Sts.ReadyForNewShuttle := FALSE;

				gBufferAreaIf.Par.ShuttleIdx := STATION_IS_EMPTY;
				IF gBufferAreaIf.Cmd.Enable THEN
					state := BUFFER_INIT;
				ELSE
					state := BUFFER_OFF;
				END_IF
			END_IF
	END_CASE;
END_PROGRAM
```

#### Init.st
```iecst
PROGRAM _INIT
	gBufferAreaIf.Par.ShuttleIdx := STATION_IS_EMPTY;
	//Define station configuration values
	gBufferAreaIf.Cfg.StationPos.X := 0.54;
	gBufferAreaIf.Cfg.StationPos.Y := 0.00; //Y value isn't used really for the buffer area

	gSysPars.BufferArea.MinBufferSize := 8;
END_PROGRAM
```

### Program Logical/Source/ProcessStations/FillStation (IEC)

#### Cyclic.st - Cyclic code
```iecst
PROGRAM _CYCLIC
	CASE state OF
		FILL_OFF: //********************************************************************************Fill station is currently disabled
			IF pFillIf.Cmd.Enable THEN
				state := FILL_INIT;
			END_IF
		FILL_INIT: //********************************************************************************Fill station is initalizing
			pFillIf.Sts.ReadyForNewShuttle := TRUE;
			pFillIf.Sts.Enabled := TRUE;
			state := FILL_WAIT_FOR_SHUTTLE;
		FILL_WAIT_FOR_SHUTTLE: //********************************************************************************Fill station is waiting for a shuttle to be present
			IF NOT pFillIf.Cmd.Enable THEN
				pFillIf.Sts.ReadyForNewShuttle := FALSE;
				pFillIf.Sts.Enabled := FALSE;
				state := FILL_OFF;
			ELSIF pFillIf.Par.ShuttleIdx <> STATION_IS_EMPTY AND pFillIf.Cmd.Process THEN
				pFillIf.Sts.ReadyForNewShuttle := FALSE;
				pFillIf.Sts.Processing := TRUE;

				FillStationFbs.FillMoveFb.Controller := ADR(gMcAcp6DController);
				FillStationFbs.FillMoveFb.ShuttleID := gShuttleIf[pFillIf.Par.ShuttleIdx].Cfg.ShuttleId;
				FillStationFbs.FillMoveFb.Mode := mcACP6D_MOVE_ABSOLUTE;
				FillStationFbs.FillMoveFb.Path := mcACP6D_PATH_Y_THEN_X;
				FillStationFbs.FillMoveFb.Velocity := stationPars.Vel;
				FillStationFbs.FillMoveFb.EndVelocity := 0;
				FillStationFbs.FillMoveFb.Acceleration := stationPars.Accel;
				FillStationFbs.FillMoveFb.PositionX := pFillIf.Cfg.StationPos.X;
				FillStationFbs.FillMoveFb.PositionY := pFillIf.Cfg.StationPos.Y;
				FillStationFbs.FillMoveFb.Execute := TRUE;

				state := FILL_ENTER_SHUTTLE;
			END_IF
		FILL_ENTER_SHUTTLE: //******************************************************************************** Fill station is moving to the filling position
			IF FillStationFbs.FillMoveFb.Error THEN
				pFillIf.Sts.Error := TRUE;

				state := FILL_ERROR;
			ELSIF FillStationFbs.FillMoveFb.Done THEN
				FillStationFbs.FillMoveFb.Execute:= FALSE;

				FillStationFbs.WaitTimer.IN := TRUE;
				FillStationFbs.WaitTimer.PT := stationPars.FillTime;

				SetupStationActions;

				state := FILL_FILLING;
			END_IF
		FILL_FILLING: //********************************************************************************Fill station is preforming the filling process
			IF FillStationFbs.WaitTimer.Q
				AND ((FillStationFbs.St1Fb.Done AND FillStationFbs.St1Fb.Execute)
				OR (FillStationFbs.St2Fb.Done AND FillStationFbs.St2Fb.Execute)
				OR (FillStationFbs.St3Fb.Done AND FillStationFbs.St3Fb.Execute)
				OR (FillStationFbs.St4Fb.Done AND FillStationFbs.St4Fb.Execute)) THEN
				FillStationFbs.WaitTimer.IN := FALSE;
				//Interface with the correct Station FB
				CASE station OF
					ST1:
						FillStationFbs.St1Fb.Execute := FALSE;
					ST2:
						FillStationFbs.St2Fb.Execute := FALSE;
					ST3:
						FillStationFbs.St3Fb.Execute := FALSE;
						macroPatternCounter := macroPatternCounter + 1;
						IF macroPatternCounter = 2 THEN
							macroPatternCounter := 0;
						END_IF
					ST4:
						FillStationFbs.St4Fb.Execute := FALSE;
				END_CASE;

				FillStationFbs.FillMoveFb.Mode := mcACP6D_MOVE_ABSOLUTE;
				FillStationFbs.FillMoveFb.Path := mcACP6D_PATH_X_THEN_Y;
				FillStationFbs.FillMoveFb.Velocity := stationPars.Vel;
				FillStationFbs.FillMoveFb.EndVelocity := 0;
				FillStationFbs.FillMoveFb.Acceleration := stationPars.Accel;
				FillStationFbs.FillMoveFb.PositionX := pFillIf.Cfg.ExitPos.X;
				FillStationFbs.FillMoveFb.PositionY := pFillIf.Cfg.ExitPos.Y;
				FillStationFbs.FillMoveFb.Execute := TRUE;

				state := FILL_EXIT_SHUTTLE;
			END_IF
		FILL_EXIT_SHUTTLE:
			IF FillStationFbs.FillMoveFb.Error THEN
				pFillIf.Sts.Error := TRUE;

				state := FILL_ERROR;
			ELSIF FillStationFbs.FillMoveFb.Acknowledge THEN
				FillStationFbs.FillMoveFb.Execute := FALSE;
				gShuttleIf[pFillIf.Par.ShuttleIdx].Cmd.NextStep := TRUE;
				pFillIf.Sts.Done := TRUE;
				pFillIf.Sts.Processing := FALSE;

				state := FILL_DONE;
			END_IF
		FILL_DONE: //********************************************************************************Fill station is done with the load process
			IF NOT pFillIf.Cmd.Enable THEN
				pFillIf.Sts.Enabled := FALSE;
				pFillIf.Sts.ReadyForNewShuttle := FALSE;
				macroPatternCounter := 0;

				state := FILL_OFF;
			ELSIF NOT pFillIf.Cmd.Process THEN
				pFillIf.Sts.Done := FALSE;

				pFillIf.Par.ShuttleIdx := STATION_IS_EMPTY;
				pFillIf.Sts.ReadyForNewShuttle := FALSE;
				pFillIf.Sts.ReadyForNewShuttle := TRUE;

				state := FILL_WAIT_FOR_SHUTTLE;
			END_IF
		FILL_ERROR: //********************************************************************************Fill station had an error
			IF pFillIf.Cmd.Reset THEN
				pFillIf.Cmd.Reset := FALSE;

				pFillIf.Par.ShuttleIdx := STATION_IS_EMPTY;

				pFillIf.Sts.Done := FALSE;
				pFillIf.Sts.Error := FALSE;
				pFillIf.Sts.Processing := FALSE;
				pFillIf.Sts.ReadyForNewShuttle := FALSE;
				pFillIf.Sts.Enabled := FALSE;

				FillStationFbs.FillMoveFb.Execute := FALSE;
				FillStationFbs.WaitTimer.IN := FALSE;

				IF pFillIf.Cmd.Enable THEN
					state := FILL_INIT;
				ELSE
					state := FILL_OFF;
				END_IF
			END_IF
	END_CASE;

	FillStationFbs.FillMoveFb();
	FillStationFbs.WaitTimer();
	//Call the appropriate station block
	CallStationFbs;

END_PROGRAM
```

#### Init.st - Init code
```iecst
PROGRAM _INIT
	ST_name(0,ADR(taskName),0);

	IF taskName = 'FillSt1' THEN
		pFillIf ACCESS ADR(gFillStationsIf[0]);
		stationPars ACCESS ADR(gSysPars.FillStations[0]);
		station := ST1;
	ELSIF taskName = 'FillSt2' THEN
		pFillIf ACCESS ADR(gFillStationsIf[1]);
		stationPars ACCESS ADR(gSysPars.FillStations[1]);
		station := ST2;
	ELSIF taskName = 'FillSt3' THEN
		pFillIf ACCESS ADR(gFillStationsIf[2]);
		stationPars ACCESS ADR(gSysPars.FillStations[2]);
		station := ST3;
	ELSIF taskName = 'FillSt4' THEN
		pFillIf ACCESS ADR(gFillStationsIf[3]);
		stationPars ACCESS ADR(gSysPars.FillStations[3]);
		station := ST4;
	END_IF

	//Absolute entrance pos
	gFillStationsIf[0].Cfg.EnterPos.X := 1.50;
	gFillStationsIf[0].Cfg.EnterPos.Y := 0.30;
	//Station center
	gFillStationsIf[0].Cfg.StationPos.X := 1.56;
	gFillStationsIf[0].Cfg.StationPos.Y := 0.12;
	//Absolute exit position
	gFillStationsIf[0].Cfg.ExitPos.X := 1.62;
	gFillStationsIf[0].Cfg.ExitPos.Y := 0.3;

	gFillStationsIf[1].Cfg.EnterPos.X := 1.98;
	gFillStationsIf[1].Cfg.EnterPos.Y := 0.3;
	gFillStationsIf[1].Cfg.StationPos.X := 2.04;
	gFillStationsIf[1].Cfg.StationPos.Y := 0.12;
	gFillStationsIf[1].Cfg.ExitPos.X := 2.1;
	gFillStationsIf[1].Cfg.ExitPos.Y := 0.3;

	gFillStationsIf[2].Cfg.ExitPos.X := 1.98;
	gFillStationsIf[2].Cfg.ExitPos.Y := 0.9;
	gFillStationsIf[2].Cfg.StationPos.X := 2.04;
	gFillStationsIf[2].Cfg.StationPos.Y := 1.08;
	gFillStationsIf[2].Cfg.EnterPos.X := 2.1;
	gFillStationsIf[2].Cfg.EnterPos.Y := 0.9;

	gFillStationsIf[3].Cfg.ExitPos.X := 1.50;
	gFillStationsIf[3].Cfg.ExitPos.Y := 0.9;
	gFillStationsIf[3].Cfg.StationPos.X := 1.56;
	gFillStationsIf[3].Cfg.StationPos.Y := 1.08;
	gFillStationsIf[3].Cfg.EnterPos.X := 1.62;
	gFillStationsIf[3].Cfg.EnterPos.Y := 0.9;

	pFillIf.Par.ShuttleIdx := STATION_IS_EMPTY;

	stationPars.Vel := 1.0;
	stationPars.Accel := 10.0;

	FillStationFbs.St1Fb.LinearVel := 0.5;// m/s
	FillStationFbs.St1Fb.ShortAxisRotVel := 1.0;//rad/s
END_PROGRAM
```

#### Types.typ - Local data types
```iecst
TYPE
	FillStationStateEnum :
		(
		FILL_OFF, (*Fill station is currently disabled*)
		FILL_INIT, (*Fill station is initalizing*)
		FILL_WAIT_FOR_SHUTTLE, (*Fill station is waiting for a shuttle to be present*)
		FILL_ENTER_SHUTTLE, (*Shuttle is entering the filling station*)
		FILL_FILLING, (*Fill station is preforming the filling process*)
		FILL_EXIT_SHUTTLE, (*Fill station is preforming the exit movement*)
		FILL_DONE, (*Fill station is done with the filling process*)
		FILL_ERROR (*Fill station had an error*)
		);
	FillStationFbTyp : 	STRUCT
		FillMoveFb : MC_BR_MoveInPlane_Acp6D;
		WaitTimer : TON;
		St1Fb : AngledMovementFb;
		St2Fb : MC_BR_MacroRun_Acp6D;
		St3Fb : WobbleMovementFb;
		St4Fb : MC_BR_MacroRun_Acp6D;
	END_STRUCT;
	FillStationEnum :
		(
		ST_UNDEF,
		ST1,
		ST2,
		ST3,
		ST4
		);
END_TYPE
```

#### Variables.var - Local variables
```iecst
VAR
	state : FillStationStateEnum;
	pFillIf : REFERENCE TO StationIfTyp;
	FillStationFbs : FillStationFbTyp;
	taskName : STRING[80];
	stationPars : REFERENCE TO FillStationParsTyp;
	station : FillStationEnum;
	macroPatternCounter : USINT;
END_VAR
```

#### LocalFunctionVars.var - Local variables
```iecst
VAR CONSTANT
	axPosX : USINT := 0;
	axPosY : USINT := 1;
	axPosZ : USINT := 2;
	axPosRX : USINT := 3;
	axPosRY : USINT := 4;
	axPosRZ : USINT := 5;
	axVel : USINT := 0;
	axVelRx : USINT := 1;
	axVelRy : USINT := 2;
	axVelRz : USINT := 3;
END_VAR
```

#### LocalFunctionsTypes.typ - Local data types
```iecst
(*Angled Movement Function block*)

TYPE
	AngledMovementInternalTyp : 	STRUCT
		state : AngledMovementInternalStateEnum;
		Fbs : AngledMovementInternalFbsTyp;
		ShPos : ARRAY[0..5]OF REAL;
		MovementNum : USINT;
	END_STRUCT;
	AngledMovementInternalFbsTyp : 	STRUCT
		Move6DFb : MC_BR_Move6D_Acp6D;
	END_STRUCT;
	AngledMovementInternalStateEnum :
		(
		ANG_INT_OFF,
		ANG_INT_MOV_WAIT,
		ANG_INT_MOV_1,
		ANG_INT_MOV_2,
		ANG_INT_MOV_3,
		ANG_INT_MOV_4,
		ANG_INT_MOV_5,
		ANG_INT_MOV_6,
		ANG_INT_MOV_7,
		ANG_INT_MOV_8,
		ANG_INT_MOV_9,
		ANG_INT_MOV_10,
		ANG_INT_DONE,
		ANG_INT_ERROR
		);
END_TYPE

(*"wobble movement function block"*)

TYPE
	WobbleMovInternalTyp : 	STRUCT
		state : WobbleMovStateEnum;
		Fbs : WobbleMovInternalFbsTyp;
	END_STRUCT;
	WobbleMovInternalFbsTyp : 	STRUCT
		VirtualMacroFb : MC_BR_MacroRun_Acp6D;
		RealMacroFb : MC_BR_MacroRun_Acp6D;
		PlanetCtrlFb : MC_BR_PlanetCtrl_Acp6D;
		StopFb : MC_BR_Stop_Acp6D;
		Move6DFb : MC_BR_Move6D_Acp6D;
	END_STRUCT;
	WobbleMovStateEnum :
		(
		WOB_INT_OFF,
		WOB_INT_SETUP_PLANET,
		WOB_INT_MACRO_RUN,
		WOB_INT_STOP,
		WOB_INT_REORIENT,
		WOB_INT_BREAK_PLANET,
		WOB_INT_DONE,
		WOB_INT_ERROR
		);
END_TYPE
```

#### LocalFunctions.fun
```iecst
{REDUND_ERROR} FUNCTION_BLOCK AngledMovementFb (*TODO: Add your comment here*) (*$GROUP=User,$CAT=User,$GROUPICON=User.png,$CATICON=User.png*)
	VAR_INPUT
		Execute : BOOL;
		Controller : REFERENCE TO McAcp6DControllerType;
		ShuttleId : USINT;
		PosStartX : REAL;
		PosStartY : REAL;
		LinearVel : REAL;
		ShortAxisRotVel : REAL;
	END_VAR
	VAR_OUTPUT
		Active : BOOL;
		Done : BOOL;
		Error : BOOL;
	END_VAR
	VAR
		Internal : AngledMovementInternalTyp;
	END_VAR
END_FUNCTION_BLOCK

{REDUND_ERROR} FUNCTION_BLOCK WobbleMovementFb (*TODO: Add your comment here*) (*$GROUP=User,$CAT=User,$GROUPICON=User.png,$CATICON=User.png*)
	VAR_INPUT
		Execute : BOOL;
		Controller : REFERENCE TO McAcp6DControllerType;
		ShuttleId : USINT;
		VirtShId : USINT;
		SunMacroID : USINT;
		PlanetMacroID : USINT;
		PosStartX : REAL;
		PosStartY : REAL;
	END_VAR
	VAR_OUTPUT
		Active : BOOL;
		Done : BOOL;
		Error : BOOL;
	END_VAR
	VAR
		Internal : WobbleMovInternalTyp;
	END_VAR
END_FUNCTION_BLOCK
```
